KUKA KRL program: EPS_2_251806_MH44A_A_20260212042239.src

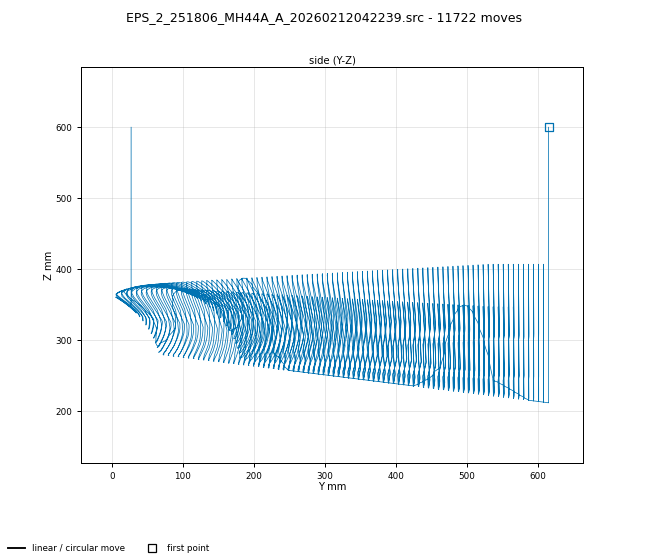
[picture p0: tool path of EPS_2_251806_MH44A_A_20260212042239.src, 11722 of 11724 moves have a stored position in this frame; points joined in program order, loops and branches not executed]
&ACCESS RVP
&REL 4
&COMMENT QRS 19112012
&PARAM EDITMASK = *
DEF PART()
EXT BAS (BAS_COMMAND :IN,REAL :IN )
INT I
BAS (#INITMOV,0 )

;KUKA QRS Post kuka4.cps  Date:22-06-2017 !

File_ID=3016

QRS_PRE_INIT()

;Init var - Until changes are made in qrs_pre_init
Outlet_Square_prg=0
Inlet_1_Square_prg=0
Inlet_2_Square_prg=0
Inlet_3_Square_prg=0
Inlet_4_Square_prg=0
Inlet_5_Square_prg=0

Outlet_1={X 0.000, Y 531.880, Z 306.500, B 0.000, E1 0.000 }
Inlet_1={X 0.000, Y 536.220, Z 246.500, B 0.000, E1 143.000 }
Outlet_1_type=201
Inlet_1_type=201
;QRS#1=Sidecore dimensions
;QRS#2=200-8" PVC SDR 35
;QRS#3=200-8" PVC SDR 35
;QRS#4=
;QRS#5=
;QRS#6=
;QRS#7=
;QRS#8=
;QRS#9=12-08 PSX
;QRS#10=12-08 PSX
;QRS#11=
;QRS#12=
;QRS#13=
;QRS#14=
;QRS#15=
;QRS#16=1220x127x686 2,25'
;QRS#17=EPS Height
;QRS#18=407
;QRS#19=*
;QRS#20= UPDATED VERSION 22-06-2017
;QRS#21=*
Outlet_Square=0100
Inlet_1_Square=0100
Inlet_2_Square=0
Inlet_3_Square=0
Inlet_4_Square=0
Inlet_5_Square=0
Mill_Square=1
Outlet_Square_Prg=204
Inlet_1_Square_prg=204

QRS_INIT()

$ADVANCE=5

; T1
PTP {E1 173.604,E2 173.604}
PTP {X 0,Y 615.501,A -85,B 0,C 180,E1 173.604,E2 173.604,E3 0,E4 0,E5 0,E6 0}
QRS_SPEED_INIT()
LIN {X 0,Y 615.501,Z 600,A -85,B 0,C 180,E1 173.604,E2 173.604,E3 0,E4 0,E5 0,E6 0} C_VEL
LIN {X 0,Y 615.501,Z 221.877,A -85,B 0,C 180,E1 173.604,E2 173.604} C_VEL
LIN {X 0,Y 615.501,Z 213.7,A -85,B 0,C 180,E1 173.604,E2 173.604} C_VEL
LIN {X 0,Y 615.484,Z 211.7,A -85,B 0,C 180,E1 173.418,E2 173.418} C_VEL
LIN {X 0,Y 615.468,Z 211.7,A -85,B 0,C 180,E1 170.802,E2 170.802} C_VEL
LIN {X 0,Y 615.482,Z 211.7,A -85,B 0,C 180,E1 168.14,E2 168.14} C_VEL
LIN {X 0,Y 615.482,Z 211.7,A -85,B 0,C 180,E1 165.452,E2 165.452} C_VEL
LIN {X 0,Y 615.471,Z 211.7,A -85,B 0,C 180,E1 162.73,E2 162.73} C_VEL
LIN {X 0,Y 615.494,Z 212.13,A -85,B 0,C 180,E1 162.045,E2 162.045} C_VEL
LIN {X 0,Y 615.475,Z 215.539,A -85,B 0,C 180,E1 159.27,E2 159.27} C_VEL
LIN {X 0,Y 615.487,Z 218.065,A -85,B 0,C 180,E1 157.157,E2 157.157} C_VEL
LIN {X 0,Y 615.458,Z 220.676,A -85,B 0,C 180,E1 155.008,E2 155.008} C_VEL
LIN {X 0,Y 615.443,Z 223.522,A -85,B 0,C 180,E1 152.822,E2 152.822} C_VEL
LIN {X 0,Y 615.473,Z 226.996,A -85,B 0,C 180,E1 150.206,E2 150.206} C_VEL
LIN {X 0,Y 615.457,Z 230.596,A -85,B 0,C 180,E1 147.542,E2 147.542} C_VEL
LIN {X 0,Y 615.42,Z 233.849,A -85,B 0,C 180,E1 145.182,E2 145.182} C_VEL
LIN {X 0,Y 615.429,Z 237.237,A -85,B 0,C 180,E1 142.756,E2 142.756} C_VEL
LIN {X 0,Y 615.465,Z 241.237,A -85,B 0,C 180,E1 139.912,E2 139.912} C_VEL
LIN {X 0,Y 615.478,Z 243.199,A -85,B 0,C 180,E1 138.54,E2 138.54} C_VEL
LIN {X 0,Y 615.494,Z 257.019,A -85,B 0,C 180,E1 138.227,E2 138.227} C_VEL
LIN {X 0,Y 615.457,Z 268.364,A -85,B 0,C 180,E1 137.852,E2 137.852} C_VEL
LIN {X 0,Y 615.434,Z 280.793,A -85,B 0,C 180,E1 137.3,E2 137.3} C_VEL
LIN {X 0,Y 615.479,Z 291.826,A -85,B 0,C 180,E1 136.662,E2 136.662} C_VEL
LIN {X 0,Y 615.498,Z 302.999,A -85,B 0,C 180,E1 135.854,E2 135.854} C_VEL
LIN {X 0,Y 615.498,Z 311.781,A -85,B 0,C 180,E1 135.067,E2 135.067} C_VEL
LIN {X 0,Y 615.498,Z 320.153,A -85,B 0,C 180,E1 134.148,E2 134.148} C_VEL
LIN {X 0,Y 615.496,Z 328.206,A -85,B 0,C 180,E1 133.051,E2 133.051} C_VEL
LIN {X 0,Y 615.494,Z 333.817,A -85,B 0,C 180,E1 132.083,E2 132.083} C_VEL
LIN {X 0,Y 615.494,Z 338.335,A -85,B 0,C 180,E1 131.098,E2 131.098} C_VEL
LIN {X 0,Y 615.495,Z 341.831,A -85,B 0,C 180,E1 130.092,E2 130.092} C_VEL
LIN {X 0,Y 615.493,Z 344.634,A -85,B 0,C 180,E1 128.903,E2 128.903} C_VEL
LIN {X 0,Y 615.496,Z 345.873,A -85,B 0,C 180,E1 128.016,E2 128.016} C_VEL
LIN {X 0,Y 615.495,Z 346.388,A -85,B 0,C 180,E1 126.94,E2 126.94} C_VEL
LIN {X 0,Y 615.492,Z 345.806,A -85,B 0,C 180,E1 125.837,E2 125.837} C_VEL
LIN {X 0,Y 615.496,Z 344.041,A -85,B 0,C 180,E1 124.705,E2 124.705} C_VEL
LIN {X 0,Y 615.494,Z 340.938,A -85,B 0,C 180,E1 123.538,E2 123.538} C_VEL
LIN {X 0,Y 615.496,Z 336.287,A -85,B 0,C 180,E1 122.335,E2 122.335} C_VEL
LIN {X 0,Y 615.496,Z 331.413,A -85,B 0,C 180,E1 121.387,E2 121.387} C_VEL
LIN {X 0,Y 615.496,Z 324.693,A -85,B 0,C 180,E1 120.348,E2 120.348} C_VEL
LIN {X 0,Y 615.497,Z 317.091,A -85,B 0,C 180,E1 119.405,E2 119.405} C_VEL
LIN {X 0,Y 615.499,Z 307.674,A -85,B 0,C 180,E1 118.456,E2 118.456} C_VEL
LIN {X 0,Y 615.498,Z 297.504,A -85,B 0,C 180,E1 117.636,E2 117.636} C_VEL
LIN {X 0,Y 615.484,Z 286.066,A -85,B 0,C 180,E1 116.897,E2 116.897} C_VEL
LIN {X 0,Y 615.481,Z 274.403,A -85,B 0,C 180,E1 116.307,E2 116.307} C_VEL
LIN {X 0,Y 615.478,Z 262.552,A -85,B 0,C 180,E1 115.852,E2 115.852} C_VEL
LIN {X 0,Y 615.493,Z 249.765,A -85,B 0,C 180,E1 115.501,E2 115.501} C_VEL
LIN {X 0,Y 615.489,Z 243.175,A -85,B 0,C 180,E1 115.355,E2 115.355} C_VEL
LIN {X 0,Y 615.482,Z 239.601,A -85,B 0,C 180,E1 112.844,E2 112.844} C_VEL
LIN {X 0,Y 615.488,Z 235.649,A -85,B 0,C 180,E1 110.032,E2 110.032} C_VEL
LIN {X 0,Y 615.466,Z 231.834,A -85,B 0,C 180,E1 107.27,E2 107.27} C_VEL
LIN {X 0,Y 615.49,Z 228.119,A -85,B 0,C 180,E1 104.548,E2 104.548} C_VEL
LIN {X 0,Y 615.457,Z 224.547,A -85,B 0,C 180,E1 101.861,E2 101.861} C_VEL
LIN {X 0,Y 615.452,Z 221.927,A -85,B 0,C 180,E1 99.862,E2 99.862} C_VEL
LIN {X 0,Y 615.444,Z 219.39,A -85,B 0,C 180,E1 97.875,E2 97.875} C_VEL
LIN {X 0,Y 615.475,Z 216.19,A -85,B 0,C 180,E1 95.241,E2 95.241} C_VEL
LIN {X 0,Y 615.47,Z 212.993,A -85,B 0,C 180,E1 92.617,E2 92.617} C_VEL
LIN {X 0,Y 615.489,Z 211.697,A -85,B 0,C 180,E1 91.308,E2 91.308} C_VEL
LIN {X 0,Y 615.487,Z 211.697,A -85,B 0,C 180,E1 88.691,E2 88.691} C_VEL
LIN {X 0,Y 615.485,Z 211.701,A -85,B 0,C 180,E1 86.071,E2 86.071} C_VEL
LIN {X 0,Y 615.493,Z 211.697,A -85,B 0,C 180,E1 83.402,E2 83.402} C_VEL
LIN {X 0,Y 615.482,Z 211.697,A -85,B 0,C 180,E1 80.8,E2 80.8} C_VEL
LIN {X 0,Y 615.484,Z 211.7,A -85,B 0,C 180,E1 78.138,E2 78.138} C_VEL
LIN {X 0,Y 615.495,Z 211.697,A -85,B 0,C 180,E1 75.45,E2 75.45} C_VEL
LIN {X 0,Y 615.472,Z 211.7,A -85,B 0,C 180,E1 72.728,E2 72.728} C_VEL
LIN {X 0,Y 615.49,Z 211.702,A -85,B 0,C 180,E1 69.967,E2 69.967} C_VEL
LIN {X 0,Y 615.486,Z 211.697,A -85,B 0,C 180,E1 67.155,E2 67.155} C_VEL
LIN {X 0,Y 615.494,Z 211.7,A -85,B 0,C 180,E1 64.284,E2 64.284} C_VEL
LIN {X 0,Y 615.49,Z 211.695,A -85,B 0,C 180,E1 61.341,E2 61.341} C_VEL
LIN {X 0,Y 615.477,Z 211.699,A -85,B 0,C 180,E1 58.912,E2 58.912} C_VEL
LIN {X 0,Y 615.479,Z 211.7,A -85,B 0,C 180,E1 56.464,E2 56.464} C_VEL
LIN {X 0,Y 615.48,Z 211.7,A -85,B 0,C 180,E1 54.165,E2 54.165} C_VEL
LIN {X 0,Y 615.477,Z 211.7,A -85,B 0,C 180,E1 51.93,E2 51.93} C_VEL
LIN {X 0,Y 615.491,Z 211.701,A -85,B 0,C 180,E1 49.393,E2 49.393} C_VEL
LIN {X 0,Y 615.475,Z 211.7,A -85,B 0,C 180,E1 46.753,E2 46.753} C_VEL
LIN {X 0,Y 615.483,Z 211.698,A -85,B 0,C 180,E1 43.996,E2 43.996} C_VEL
LIN {X 0,Y 615.494,Z 211.698,A -85,B 0,C 180,E1 41.471,E2 41.471} C_VEL
LIN {X 0,Y 615.487,Z 211.7,A -85,B 0,C 180,E1 38.902,E2 38.902} C_VEL
LIN {X 0,Y 615.498,Z 211.696,A -85,B 0,C 180,E1 35.834,E2 35.834} C_VEL
LIN {X 0,Y 615.488,Z 211.701,A -85,B 0,C 180,E1 33.234,E2 33.234} C_VEL
LIN {X 0,Y 615.484,Z 211.701,A -85,B 0,C 180,E1 30.918,E2 30.918} C_VEL
LIN {X 0,Y 615.486,Z 211.698,A -85,B 0,C 180,E1 28.449,E2 28.449} C_VEL
LIN {X 0,Y 615.488,Z 211.698,A -85,B 0,C 180,E1 25.568,E2 25.568} C_VEL
LIN {X 0,Y 615.486,Z 211.7,A -85,B 0,C 180,E1 22.843,E2 22.843} C_VEL
LIN {X 0,Y 615.495,Z 211.695,A -85,B 0,C 180,E1 20.031,E2 20.031} C_VEL
LIN {X 0,Y 615.497,Z 211.7,A -85,B 0,C 180,E1 17.269,E2 17.269} C_VEL
LIN {X 0,Y 615.488,Z 211.696,A -85,B 0,C 180,E1 14.548,E2 14.548} C_VEL
LIN {X 0,Y 615.488,Z 211.698,A -85,B 0,C 180,E1 11.86,E2 11.86} C_VEL
LIN {X 0,Y 615.493,Z 211.7,A -85,B 0,C 180,E1 9.198,E2 9.198} C_VEL
LIN {X 0,Y 615.493,Z 211.695,A -85,B 0,C 180,E1 6.555,E2 6.555} C_VEL
LIN {X 0,Y 615.483,Z 211.698,A -85,B 0,C 180,E1 3.927,E2 3.927} C_VEL
LIN {X 0,Y 615.491,Z 211.701,A -85,B 0,C 180,E1 1.308,E2 1.308} C_VEL
LIN {X 0,Y 615.495,Z 211.696,A -85,B 0,C 180,E1 -1.31,E2 -1.31} C_VEL
LIN {X 0,Y 615.477,Z 211.698,A -85,B 0,C 180,E1 -3.93,E2 -3.93} C_VEL
LIN {X 0,Y 615.482,Z 211.701,A -85,B 0,C 180,E1 -6.569,E2 -6.569} C_VEL
LIN {X 0,Y 615.496,Z 211.697,A -85,B 0,C 180,E1 -9.2,E2 -9.2} C_VEL
LIN {X 0,Y 615.47,Z 211.7,A -85,B 0,C 180,E1 -11.862,E2 -11.862} C_VEL
LIN {X 0,Y 615.478,Z 211.701,A -85,B 0,C 180,E1 -14.55,E2 -14.55} C_VEL
LIN {X 0,Y 615.493,Z 211.697,A -85,B 0,C 180,E1 -17.271,E2 -17.271} C_VEL
LIN {X 0,Y 615.47,Z 211.7,A -85,B 0,C 180,E1 -20.034,E2 -20.034} C_VEL
LIN {X 0,Y 615.497,Z 211.699,A -85,B 0,C 180,E1 -22.845,E2 -22.845} C_VEL
LIN {X 0,Y 615.471,Z 211.7,A -85,B 0,C 180,E1 -25.717,E2 -25.717} C_VEL
LIN {X 0,Y 615.494,Z 211.701,A -85,B 0,C 180,E1 -28.45,E2 -28.45} C_VEL
LIN {X 0,Y 615.487,Z 211.697,A -85,B 0,C 180,E1 -31.085,E2 -31.085} C_VEL
LIN {X 0,Y 615.484,Z 211.7,A -85,B 0,C 180,E1 -34.023,E2 -34.023} C_VEL
LIN {X 0,Y 615.49,Z 211.696,A -85,B 0,C 180,E1 -36.936,E2 -36.936} C_VEL
LIN {X 0,Y 615.484,Z 211.7,A -85,B 0,C 180,E1 -39.751,E2 -39.751} C_VEL
LIN {X 0,Y 615.494,Z 211.698,A -85,B 0,C 180,E1 -42.353,E2 -42.353} C_VEL
LIN {X 0,Y 615.483,Z 211.697,A -85,B 0,C 180,E1 -45.07,E2 -45.07} C_VEL
LIN {X 0,Y 615.493,Z 211.701,A -85,B 0,C 180,E1 -47.92,E2 -47.92} C_VEL
LIN {X 0,Y 615.489,Z 211.696,A -85,B 0,C 180,E1 -50.938,E2 -50.938} C_VEL
LIN {X 0,Y 615.486,Z 211.701,A -85,B 0,C 180,E1 -53.574,E2 -53.574} C_VEL
LIN {X 0,Y 615.49,Z 211.764,A -85,B 0,C 180,E1 -54.484,E2 -54.484} C_VEL
LIN {X 0,Y 615.478,Z 220.56,A -85,B 0,C 180,E1 -57.153,E2 -57.153} C_VEL
LIN {X 0,Y 615.476,Z 228.497,A -85,B 0,C 180,E1 -59.46,E2 -59.46} C_VEL
LIN {X 0,Y 615.451,Z 237.756,A -85,B 0,C 180,E1 -62.082,E2 -62.082} C_VEL
LIN {X 0,Y 615.464,Z 247.261,A -85,B 0,C 180,E1 -64.718,E2 -64.718} C_VEL
LIN {X 0,Y 615.448,Z 256.24,A -85,B 0,C 180,E1 -67.153,E2 -67.153} C_VEL
LIN {X 0,Y 615.478,Z 264.815,A -85,B 0,C 180,E1 -69.446,E2 -69.446} C_VEL
LIN {X 0,Y 615.492,Z 276.01,A -85,B 0,C 180,E1 -72.386,E2 -72.386} C_VEL
LIN {X 0,Y 615.484,Z 286.539,A -85,B 0,C 180,E1 -75.112,E2 -75.112} C_VEL
LIN {X 0,Y 615.465,Z 297.082,A -85,B 0,C 180,E1 -77.804,E2 -77.804} C_VEL
LIN {X 0,Y 615.496,Z 299.207,A -85,B 0,C 180,E1 -78.348,E2 -78.348} C_VEL
LIN {X 0,Y 615.497,Z 313.797,A -85,B 0,C 180,E1 -78.64,E2 -78.64} C_VEL
LIN {X 0,Y 615.455,Z 326.947,A -85,B 0,C 180,E1 -79.05,E2 -79.05} C_VEL
LIN {X 0,Y 615.447,Z 338.759,A -85,B 0,C 180,E1 -79.555,E2 -79.555} C_VEL
LIN {X 0,Y 615.497,Z 349.375,A -85,B 0,C 180,E1 -80.137,E2 -80.137} C_VEL
LIN {X 0,Y 615.498,Z 360.223,A -85,B 0,C 180,E1 -80.884,E2 -80.884} C_VEL
LIN {X 0,Y 615.497,Z 370.805,A -85,B 0,C 180,E1 -81.793,E2 -81.793} C_VEL
LIN {X 0,Y 615.498,Z 378.6,A -85,B 0,C 180,E1 -82.619,E2 -82.619} C_VEL
LIN {X 0,Y 615.496,Z 386.198,A -85,B 0,C 180,E1 -83.607,E2 -83.607} C_VEL
LIN {X 0,Y 615.498,Z 393.201,A -85,B 0,C 180,E1 -84.758,E2 -84.758} C_VEL
LIN {X 0,Y 615.494,Z 397.848,A -85,B 0,C 180,E1 -85.743,E2 -85.743} C_VEL
LIN {X 0,Y 615.494,Z 401.397,A -85,B 0,C 180,E1 -86.726,E2 -86.726} C_VEL
LIN {X 0,Y 615.497,Z 403.231,A -85,B 0,C 180,E1 -87.382,E2 -87.382} C_VEL
LIN {X 0,Y 615.5,Z 404.606,A -85,B 0,C 180,E1 -88.036,E2 -88.036} C_VEL
LIN {X 0,Y 615.496,Z 406.173,A -85,B 0,C 180,E1 -89.345,E2 -89.345} C_VEL
LIN {X 0,Y 615.494,Z 406.389,A -85,B 0,C 180,E1 -89.999,E2 -89.999} C_VEL
LIN {X 0,Y 615.495,Z 405.581,A -85,B 0,C 180,E1 -91.308,E2 -91.308} C_VEL
LIN {X 0,Y 615.5,Z 404.609,A -85,B 0,C 180,E1 -91.962,E2 -91.962} C_VEL
LIN {X 0,Y 615.497,Z 403.235,A -85,B 0,C 180,E1 -92.617,E2 -92.617} C_VEL
LIN {X 0,Y 615.496,Z 400.352,A -85,B 0,C 180,E1 -93.6,E2 -93.6} C_VEL
LIN {X 0,Y 615.498,Z 396.444,A -85,B 0,C 180,E1 -94.584,E2 -94.584} C_VEL
LIN {X 0,Y 615.499,Z 391.409,A -85,B 0,C 180,E1 -95.569,E2 -95.569} C_VEL
LIN {X 0,Y 615.497,Z 384.871,A -85,B 0,C 180,E1 -96.583,E2 -96.583} C_VEL
LIN {X 0,Y 615.497,Z 377.139,A -85,B 0,C 180,E1 -97.545,E2 -97.545} C_VEL
LIN {X 0,Y 615.498,Z 369.052,A -85,B 0,C 180,E1 -98.37,E2 -98.37} C_VEL
LIN {X 0,Y 615.499,Z 359.177,A -85,B 0,C 180,E1 -99.198,E2 -99.198} C_VEL
LIN {X 0,Y 615.486,Z 347.993,A -85,B 0,C 180,E1 -99.945,E2 -99.945} C_VEL
LIN {X 0,Y 615.445,Z 337.044,A -85,B 0,C 180,E1 -100.527,E2 -100.527} C_VEL
LIN {X 0,Y 615.461,Z 324.771,A -85,B 0,C 180,E1 -101.031,E2 -101.031} C_VEL
LIN {X 0,Y 615.498,Z 312.093,A -85,B 0,C 180,E1 -101.401,E2 -101.401} C_VEL
LIN {X 0,Y 615.496,Z 299.212,A -85,B 0,C 180,E1 -101.651,E2 -101.651} C_VEL
LIN {X 0,Y 615.469,Z 289.073,A -85,B 0,C 180,E1 -104.24,E2 -104.24} C_VEL
LIN {X 0,Y 615.484,Z 278.644,A -85,B 0,C 180,E1 -106.928,E2 -106.928} C_VEL
LIN {X 0,Y 615.487,Z 268.104,A -85,B 0,C 180,E1 -109.684,E2 -109.684} C_VEL
LIN {X 0,Y 615.474,Z 258.107,A -85,B 0,C 180,E1 -112.342,E2 -112.342} C_VEL
LIN {X 0,Y 615.442,Z 248.325,A -85,B 0,C 180,E1 -114.993,E2 -114.993} C_VEL
LIN {X 0,Y 615.492,Z 239.078,A -85,B 0,C 180,E1 -117.544,E2 -117.544} C_VEL
LIN {X 0,Y 615.459,Z 229.832,A -85,B 0,C 180,E1 -120.161,E2 -120.161} C_VEL
LIN {X 0,Y 615.486,Z 221.872,A -85,B 0,C 180,E1 -122.457,E2 -122.457} C_VEL
LIN {X 0,Y 615.491,Z 212.793,A -85,B 0,C 180,E1 -125.213,E2 -125.213} C_VEL
LIN {X 0,Y 615.486,Z 211.697,A -85,B 0,C 180,E1 -125.615,E2 -125.615} C_VEL
LIN {X 0,Y 615.469,Z 211.7,A -85,B 0,C 180,E1 -128.069,E2 -128.069} C_VEL
LIN {X 0,Y 615.474,Z 211.701,A -85,B 0,C 180,E1 -130.607,E2 -130.607} C_VEL
LIN {X 0,Y 615.499,Z 211.698,A -85,B 0,C 180,E1 -133.243,E2 -133.243} C_VEL
LIN {X 0,Y 615.469,Z 211.7,A -85,B 0,C 180,E1 -136.003,E2 -136.003} C_VEL
LIN {X 0,Y 615.476,Z 211.7,A -85,B 0,C 180,E1 -138.525,E2 -138.525} C_VEL
LIN {X 0,Y 615.494,Z 211.701,A -85,B 0,C 180,E1 -141.095,E2 -141.095} C_VEL
LIN {X 0,Y 615.48,Z 211.7,A -85,B 0,C 180,E1 -143.574,E2 -143.574} C_VEL
LIN {X 0,Y 615.474,Z 211.7,A -85,B 0,C 180,E1 -145.976,E2 -145.976} C_VEL
LIN {X 0,Y 615.472,Z 211.7,A -85,B 0,C 180,E1 -148.313,E2 -148.313} C_VEL
LIN {X 0,Y 615.484,Z 211.697,A -85,B 0,C 180,E1 -150.593,E2 -150.593} C_VEL
LIN {X 0,Y 615.492,Z 211.702,A -85,B 0,C 180,E1 -153.555,E2 -153.555} C_VEL
LIN {X 0,Y 615.485,Z 211.7,A -85,B 0,C 180,E1 -155.99,E2 -155.99} C_VEL
LIN {X 0,Y 615.485,Z 211.697,A -85,B 0,C 180,E1 -158.567,E2 -158.567} C_VEL
LIN {X 0,Y 615.495,Z 211.699,A -85,B 0,C 180,E1 -161.391,E2 -161.391} C_VEL
LIN {X 0,Y 615.478,Z 211.699,A -85,B 0,C 180,E1 -164.094,E2 -164.094} C_VEL
LIN {X 0,Y 615.498,Z 211.695,A -85,B 0,C 180,E1 -166.798,E2 -166.798} C_VEL
LIN {X 0,Y 615.487,Z 211.702,A -85,B 0,C 180,E1 -169.472,E2 -169.472} C_VEL
LIN {X 0,Y 615.479,Z 211.698,A -85,B 0,C 180,E1 -172.123,E2 -172.123} C_VEL
LIN {X 0,Y 615.495,Z 211.696,A -85,B 0,C 180,E1 -174.758,E2 -174.758} C_VEL
LIN {X 0,Y 615.489,Z 211.701,A -85,B 0,C 180,E1 -177.381,E2 -177.381} C_VEL
LIN {X 0,Y 615.482,Z 211.698,A -85,B 0,C 180,E1 -179.999,E2 -179.999} C_VEL
LIN {X 0,Y 615.494,Z 211.695,A -85,B 0,C 180,E1 -182.617,E2 -182.617} C_VEL
LIN {X 0,Y 615.496,Z 211.7,A -85,B 0,C 180,E1 -185.24,E2 -185.24} C_VEL
LIN {X 0,Y 615.484,Z 211.7,A -85,B 0,C 180,E1 -186.582,E2 -186.582} C_VEL
LIN {X 0,Y 614.8,Z 211.847,A -85,B 0,C 180,E1 -187.128,E2 -187.128} C_VEL
LIN {X 0,Y 611.954,Z 212.259,A -85,B 0,C 180,E1 -188.014,E2 -188.014} C_VEL
LIN {X 0,Y 609.562,Z 212.568,A -85,B 0,C 180,E1 -188.727,E2 -188.727} C_VEL
LIN {X 0,Y 608.536,Z 212.685,A -85,B 0,C 180,E1 -189.276,E2 -189.276} C_VEL
LIN {X 0,Y 608.452,Z 212.694,A -85,B 0,C 180,E1 -189.463,E2 -189.463} C_VEL
LIN {X 0,Y 608.458,Z 212.697,A -85,B 0,C 180,E1 -191.999,E2 -191.999} C_VEL
LIN {X 0,Y 608.469,Z 212.693,A -85,B 0,C 180,E1 -194.719,E2 -194.719} C_VEL
LIN {X 0,Y 608.445,Z 212.697,A -85,B 0,C 180,E1 -197.475,E2 -197.475} C_VEL
LIN {X 0,Y 608.42,Z 214.125,A -85,B 0,C 180,E1 -198.869,E2 -198.869} C_VEL
LIN {X 0,Y 608.441,Z 217.534,A -85,B 0,C 180,E1 -201.691,E2 -201.691} C_VEL
LIN {X 0,Y 608.446,Z 220.984,A -85,B 0,C 180,E1 -204.57,E2 -204.57} C_VEL
LIN {X 0,Y 608.391,Z 224.301,A -85,B 0,C 180,E1 -207.193,E2 -207.193} C_VEL
LIN {X 0,Y 608.445,Z 227.967,A -85,B 0,C 180,E1 -209.969,E2 -209.969} C_VEL
LIN {X 0,Y 608.386,Z 231.902,A -85,B 0,C 180,E1 -212.882,E2 -212.882} C_VEL
LIN {X 0,Y 608.375,Z 235.196,A -85,B 0,C 180,E1 -215.28,E2 -215.28} C_VEL
LIN {X 0,Y 608.38,Z 239.308,A -85,B 0,C 180,E1 -218.231,E2 -218.231} C_VEL
LIN {X 0,Y 608.384,Z 242.257,A -85,B 0,C 180,E1 -220.323,E2 -220.323} C_VEL
LIN {X 0,Y 608.398,Z 243.686,A -85,B 0,C 180,E1 -221.33,E2 -221.33} C_VEL
LIN {X 0,Y 608.546,Z 257.819,A -85,B 0,C 180,E1 -221.662,E2 -221.662} C_VEL
LIN {X 0,Y 608.477,Z 269.465,A -85,B 0,C 180,E1 -222.058,E2 -222.058} C_VEL
LIN {X 0,Y 608.448,Z 281.581,A -85,B 0,C 180,E1 -222.614,E2 -222.614} C_VEL
LIN {X 0,Y 608.482,Z 293.339,A -85,B 0,C 180,E1 -223.311,E2 -223.311} C_VEL
LIN {X 0,Y 608.471,Z 303.546,A -85,B 0,C 180,E1 -224.066,E2 -224.066} C_VEL
LIN {X 0,Y 608.458,Z 313.645,A -85,B 0,C 180,E1 -224.999,E2 -224.999} C_VEL
LIN {X 0,Y 608.465,Z 321.852,A -85,B 0,C 180,E1 -225.932,E2 -225.932} C_VEL
LIN {X 0,Y 608.448,Z 328.559,A -85,B 0,C 180,E1 -226.867,E2 -226.867} C_VEL
LIN {X 0,Y 608.429,Z 334.694,A -85,B 0,C 180,E1 -227.937,E2 -227.937} C_VEL
LIN {X 0,Y 608.43,Z 338.727,A -85,B 0,C 180,E1 -228.822,E2 -228.822} C_VEL
LIN {X 0,Y 608.434,Z 343.095,A -85,B 0,C 180,E1 -230.129,E2 -230.129} C_VEL
LIN {X 0,Y 608.414,Z 345.782,A -85,B 0,C 180,E1 -231.409,E2 -231.409} C_VEL
LIN {X 0,Y 608.425,Z 346.691,A -85,B 0,C 180,E1 -232.251,E2 -232.251} C_VEL
LIN {X 0,Y 608.43,Z 346.997,A -85,B 0,C 180,E1 -233.084,E2 -233.084} C_VEL
LIN {X 0,Y 608.441,Z 346.611,A -85,B 0,C 180,E1 -233.953,E2 -233.953} C_VEL
LIN {X 0,Y 608.423,Z 345.094,A -85,B 0,C 180,E1 -235.095,E2 -235.095} C_VEL
LIN {X 0,Y 608.434,Z 342.044,A -85,B 0,C 180,E1 -236.328,E2 -236.328} C_VEL
LIN {X 0,Y 608.428,Z 337.821,A -85,B 0,C 180,E1 -237.479,E2 -237.479} C_VEL
LIN {X 0,Y 608.444,Z 331.846,A -85,B 0,C 180,E1 -238.683,E2 -238.683} C_VEL
LIN {X 0,Y 608.444,Z 324.771,A -85,B 0,C 180,E1 -239.772,E2 -239.772} C_VEL
LIN {X 0,Y 608.45,Z 316.476,A -85,B 0,C 180,E1 -240.791,E2 -240.791} C_VEL
LIN {X 0,Y 608.467,Z 306.911,A -85,B 0,C 180,E1 -241.735,E2 -241.735} C_VEL
LIN {X 0,Y 608.493,Z 296.237,A -85,B 0,C 180,E1 -242.58,E2 -242.58} C_VEL
LIN {X 0,Y 608.481,Z 286.114,A -85,B 0,C 180,E1 -243.228,E2 -243.228} C_VEL
LIN {X 0,Y 608.494,Z 274.258,A -85,B 0,C 180,E1 -243.829,E2 -243.829} C_VEL
LIN {X 0,Y 608.522,Z 261.978,A -85,B 0,C 180,E1 -244.3,E2 -244.3} C_VEL
LIN {X 0,Y 608.536,Z 249.165,A -85,B 0,C 180,E1 -244.648,E2 -244.648} C_VEL
LIN {X 0,Y 608.422,Z 243.676,A -85,B 0,C 180,E1 -244.767,E2 -244.767} C_VEL
LIN {X 0,Y 608.416,Z 239.68,A -85,B 0,C 180,E1 -247.593,E2 -247.593} C_VEL
LIN {X 0,Y 608.402,Z 235.722,A -85,B 0,C 180,E1 -250.428,E2 -250.428} C_VEL
LIN {X 0,Y 608.436,Z 231.888,A -85,B 0,C 180,E1 -253.216,E2 -253.216} C_VEL
LIN {X 0,Y 608.421,Z 228.138,A -85,B 0,C 180,E1 -255.994,E2 -255.994} C_VEL
LIN {X 0,Y 608.395,Z 224.591,A -85,B 0,C 180,E1 -258.675,E2 -258.675} C_VEL
LIN {X 0,Y 608.454,Z 221.141,A -85,B 0,C 180,E1 -261.365,E2 -261.365} C_VEL
LIN {X 0,Y 608.381,Z 217.909,A -85,B 0,C 180,E1 -264.033,E2 -264.033} C_VEL
LIN {X 0,Y 608.435,Z 214.682,A -85,B 0,C 180,E1 -266.69,E2 -266.69} C_VEL
LIN {X 0,Y 608.439,Z 213.067,A -85,B 0,C 180,E1 -268.015,E2 -268.015} C_VEL
LIN {X 0,Y 608.484,Z 212.693,A -85,B 0,C 180,E1 -269.339,E2 -269.339} C_VEL
LIN {X 0,Y 608.451,Z 212.696,A -85,B 0,C 180,E1 -271.986,E2 -271.986} C_VEL
LIN {X 0,Y 608.448,Z 212.695,A -85,B 0,C 180,E1 -274.638,E2 -274.638} C_VEL
LIN {X 0,Y 608.48,Z 212.693,A -85,B 0,C 180,E1 -277.3,E2 -277.3} C_VEL
LIN {X 0,Y 608.458,Z 212.695,A -85,B 0,C 180,E1 -279.978,E2 -279.978} C_VEL
LIN {X 0,Y 608.477,Z 212.692,A -85,B 0,C 180,E1 -282.678,E2 -282.678} C_VEL
LIN {X 0,Y 608.468,Z 212.696,A -85,B 0,C 180,E1 -285.407,E2 -285.407} C_VEL
LIN {X 0,Y 608.451,Z 212.695,A -85,B 0,C 180,E1 -288.172,E2 -288.172} C_VEL
LIN {X 0,Y 608.455,Z 212.696,A -85,B 0,C 180,E1 -290.982,E2 -290.982} C_VEL
LIN {X 0,Y 608.448,Z 212.696,A -85,B 0,C 180,E1 -293.125,E2 -293.125} C_VEL
LIN {X 0,Y 608.451,Z 212.696,A -85,B 0,C 180,E1 -296.036,E2 -296.036} C_VEL
LIN {X 0,Y 608.477,Z 212.692,A -85,B 0,C 180,E1 -298.624,E2 -298.624} C_VEL
LIN {X 0,Y 608.468,Z 212.694,A -85,B 0,C 180,E1 -301.317,E2 -301.317} C_VEL
LIN {X 0,Y 608.468,Z 212.696,A -85,B 0,C 180,E1 -303.737,E2 -303.737} C_VEL
LIN {X 0,Y 608.471,Z 212.696,A -85,B 0,C 180,E1 -306.091,E2 -306.091} C_VEL
LIN {X 0,Y 608.456,Z 212.696,A -85,B 0,C 180,E1 -308.59,E2 -308.59} C_VEL
LIN {X 0,Y 608.45,Z 212.695,A -85,B 0,C 180,E1 -311.343,E2 -311.343} C_VEL
LIN {X 0,Y 608.465,Z 212.695,A -85,B 0,C 180,E1 -314.267,E2 -314.267} C_VEL
LIN {X 0,Y 608.436,Z 212.697,A -85,B 0,C 180,E1 -317.041,E2 -317.041} C_VEL
LIN {X 0,Y 608.45,Z 212.697,A -85,B 0,C 180,E1 -319.698,E2 -319.698} C_VEL
LIN {X 0,Y 608.462,Z 212.696,A -85,B 0,C 180,E1 -322.255,E2 -322.255} C_VEL
LIN {X 0,Y 608.442,Z 212.697,A -85,B 0,C 180,E1 -324.724,E2 -324.724} C_VEL
LIN {X 0,Y 608.455,Z 212.695,A -85,B 0,C 180,E1 -327.122,E2 -327.122} C_VEL
LIN {X 0,Y 608.47,Z 212.695,A -85,B 0,C 180,E1 -330.029,E2 -330.029} C_VEL
LIN {X 0,Y 608.467,Z 212.693,A -85,B 0,C 180,E1 -332.796,E2 -332.796} C_VEL
LIN {X 0,Y 608.449,Z 212.695,A -85,B 0,C 180,E1 -335.43,E2 -335.43} C_VEL
LIN {X 0,Y 608.464,Z 212.695,A -85,B 0,C 180,E1 -338.31,E2 -338.31} C_VEL
LIN {X 0,Y 608.454,Z 212.695,A -85,B 0,C 180,E1 -341.132,E2 -341.132} C_VEL
LIN {X 0,Y 608.456,Z 212.697,A -85,B 0,C 180,E1 -343.907,E2 -343.907} C_VEL
LIN {X 0,Y 608.455,Z 212.694,A -85,B 0,C 180,E1 -346.645,E2 -346.645} C_VEL
LIN {X 0,Y 608.463,Z 212.695,A -85,B 0,C 180,E1 -349.351,E2 -349.351} C_VEL
LIN {X 0,Y 608.473,Z 212.694,A -85,B 0,C 180,E1 -352.034,E2 -352.034} C_VEL
LIN {X 0,Y 608.451,Z 212.695,A -85,B 0,C 180,E1 -354.699,E2 -354.699} C_VEL
LIN {X 0,Y 608.478,Z 212.693,A -85,B 0,C 180,E1 -357.353,E2 -357.353} C_VEL
LIN {X 0,Y 608.478,Z 212.694,A -85,B 0,C 180,E1 -360.001,E2 -360.001} C_VEL
LIN {X 0,Y 608.465,Z 212.693,A -85,B 0,C 180,E1 -362.649,E2 -362.649} C_VEL
LIN {X 0,Y 608.466,Z 212.694,A -85,B 0,C 180,E1 -365.303,E2 -365.303} C_VEL
LIN {X 0,Y 608.479,Z 212.694,A -85,B 0,C 180,E1 -367.968,E2 -367.968} C_VEL
LIN {X 0,Y 608.451,Z 212.695,A -85,B 0,C 180,E1 -370.651,E2 -370.651} C_VEL
LIN {X 0,Y 608.469,Z 212.694,A -85,B 0,C 180,E1 -373.357,E2 -373.357} C_VEL
LIN {X 0,Y 608.456,Z 212.696,A -85,B 0,C 180,E1 -376.095,E2 -376.095} C_VEL
LIN {X 0,Y 608.456,Z 212.694,A -85,B 0,C 180,E1 -378.87,E2 -378.87} C_VEL
LIN {X 0,Y 608.469,Z 212.695,A -85,B 0,C 180,E1 -381.692,E2 -381.692} C_VEL
LIN {X 0,Y 608.451,Z 212.695,A -85,B 0,C 180,E1 -384.572,E2 -384.572} C_VEL
LIN {X 0,Y 608.489,Z 212.692,A -85,B 0,C 180,E1 -387.208,E2 -387.208} C_VEL
LIN {X 0,Y 608.445,Z 212.696,A -85,B 0,C 180,E1 -389.967,E2 -389.967} C_VEL
LIN {X 0,Y 608.453,Z 212.695,A -85,B 0,C 180,E1 -392.52,E2 -392.52} C_VEL
LIN {X 0,Y 608.442,Z 212.699,A -85,B 0,C 180,E1 -395.278,E2 -395.278} C_VEL
LIN {X 0,Y 608.463,Z 212.696,A -85,B 0,C 180,E1 -397.747,E2 -397.747} C_VEL
LIN {X 0,Y 608.451,Z 212.695,A -85,B 0,C 180,E1 -400.328,E2 -400.328} C_VEL
LIN {X 0,Y 608.482,Z 212.694,A -85,B 0,C 180,E1 -403.309,E2 -403.309} C_VEL
LIN {X 0,Y 608.465,Z 212.693,A -85,B 0,C 180,E1 -406.129,E2 -406.129} C_VEL
LIN {X 0,Y 608.464,Z 212.694,A -85,B 0,C 180,E1 -408.823,E2 -408.823} C_VEL
LIN {X 0,Y 608.457,Z 212.695,A -85,B 0,C 180,E1 -411.762,E2 -411.762} C_VEL
LIN {X 0,Y 608.476,Z 212.766,A -85,B 0,C 180,E1 -414.317,E2 -414.317} C_VEL
LIN {X 0,Y 608.521,Z 220.56,A -85,B 0,C 180,E1 -416.729,E2 -416.729} C_VEL
LIN {X 0,Y 608.502,Z 229.822,A -85,B 0,C 180,E1 -419.456,E2 -419.456} C_VEL
LIN {X 0,Y 608.469,Z 239.125,A -85,B 0,C 180,E1 -422.109,E2 -422.109} C_VEL
LIN {X 0,Y 608.454,Z 248.392,A -85,B 0,C 180,E1 -424.698,E2 -424.698} C_VEL
LIN {X 0,Y 608.465,Z 258.723,A -85,B 0,C 180,E1 -427.523,E2 -427.523} C_VEL
LIN {X 0,Y 608.457,Z 269.574,A -85,B 0,C 180,E1 -430.429,E2 -430.429} C_VEL
LIN {X 0,Y 608.452,Z 280.166,A -85,B 0,C 180,E1 -433.215,E2 -433.215} C_VEL
LIN {X 0,Y 608.443,Z 290.884,A -85,B 0,C 180,E1 -435.994,E2 -435.994} C_VEL
LIN {X 0,Y 608.443,Z 299.528,A -85,B 0,C 180,E1 -438.211,E2 -438.211} C_VEL
LIN {X 0,Y 608.545,Z 314.673,A -85,B 0,C 180,E1 -438.529,E2 -438.529} C_VEL
LIN {X 0,Y 608.478,Z 327.497,A -85,B 0,C 180,E1 -438.939,E2 -438.939} C_VEL
LIN {X 0,Y 608.474,Z 338.908,A -85,B 0,C 180,E1 -439.434,E2 -439.434} C_VEL
LIN {X 0,Y 608.486,Z 349.568,A -85,B 0,C 180,E1 -440.023,E2 -440.023} C_VEL
LIN {X 0,Y 608.483,Z 360.466,A -85,B 0,C 180,E1 -440.778,E2 -440.778} C_VEL
LIN {X 0,Y 608.475,Z 371.105,A -85,B 0,C 180,E1 -441.698,E2 -441.698} C_VEL
LIN {X 0,Y 608.471,Z 378.955,A -85,B 0,C 180,E1 -442.533,E2 -442.533} C_VEL
LIN {X 0,Y 608.461,Z 386.285,A -85,B 0,C 180,E1 -443.484,E2 -443.484} C_VEL
LIN {X 0,Y 608.451,Z 391.862,A -85,B 0,C 180,E1 -444.365,E2 -444.365} C_VEL
LIN {X 0,Y 608.432,Z 396.947,A -85,B 0,C 180,E1 -445.362,E2 -445.362} C_VEL
LIN {X 0,Y 608.449,Z 400.894,A -85,B 0,C 180,E1 -446.357,E2 -446.357} C_VEL
LIN {X 0,Y 608.425,Z 403.807,A -85,B 0,C 180,E1 -447.351,E2 -447.351} C_VEL
LIN {X 0,Y 608.445,Z 405.2,A -85,B 0,C 180,E1 -448.014,E2 -448.014} C_VEL
LIN {X 0,Y 608.438,Z 406.783,A -85,B 0,C 180,E1 -449.338,E2 -449.338} C_VEL
LIN {X 0,Y 608.434,Z 407,A -85,B 0,C 180,E1 -449.999,E2 -449.999} C_VEL
LIN {X 0,Y 608.448,Z 406.185,A -85,B 0,C 180,E1 -451.323,E2 -451.323} C_VEL
LIN {X 0,Y 608.445,Z 405.202,A -85,B 0,C 180,E1 -451.985,E2 -451.985} C_VEL
LIN {X 0,Y 608.425,Z 403.811,A -85,B 0,C 180,E1 -452.648,E2 -452.648} C_VEL
LIN {X 0,Y 608.449,Z 400.898,A -85,B 0,C 180,E1 -453.642,E2 -453.642} C_VEL
LIN {X 0,Y 608.432,Z 396.953,A -85,B 0,C 180,E1 -454.637,E2 -454.637} C_VEL
LIN {X 0,Y 608.438,Z 390.881,A -85,B 0,C 180,E1 -455.8,E2 -455.8} C_VEL
LIN {X 0,Y 608.462,Z 384.24,A -85,B 0,C 180,E1 -456.799,E2 -456.799} C_VEL
LIN {X 0,Y 608.456,Z 375.995,A -85,B 0,C 180,E1 -457.8,E2 -457.8} C_VEL
LIN {X 0,Y 608.472,Z 367.544,A -85,B 0,C 180,E1 -458.635,E2 -458.635} C_VEL
LIN {X 0,Y 608.481,Z 357.1,A -85,B 0,C 180,E1 -459.473,E2 -459.473} C_VEL
LIN {X 0,Y 608.494,Z 346.767,A -85,B 0,C 180,E1 -460.144,E2 -460.144} C_VEL
LIN {X 0,Y 608.469,Z 335.851,A -85,B 0,C 180,E1 -460.713,E2 -460.713} C_VEL
LIN {X 0,Y 608.493,Z 324.095,A -85,B 0,C 180,E1 -461.186,E2 -461.186} C_VEL
LIN {X 0,Y 608.549,Z 311.297,A -85,B 0,C 180,E1 -461.554,E2 -461.554} C_VEL
LIN {X 0,Y 608.443,Z 299.533,A -85,B 0,C 180,E1 -461.788,E2 -461.788} C_VEL
LIN {X 0,Y 608.435,Z 289.438,A -85,B 0,C 180,E1 -464.379,E2 -464.379} C_VEL
LIN {X 0,Y 608.442,Z 278.847,A -85,B 0,C 180,E1 -467.13,E2 -467.13} C_VEL
LIN {X 0,Y 608.457,Z 269.58,A -85,B 0,C 180,E1 -469.57,E2 -469.57} C_VEL
LIN {X 0,Y 608.46,Z 258.728,A -85,B 0,C 180,E1 -472.476,E2 -472.476} C_VEL
LIN {X 0,Y 608.454,Z 248.398,A -85,B 0,C 180,E1 -475.3,E2 -475.3} C_VEL
LIN {X 0,Y 608.468,Z 239.13,A -85,B 0,C 180,E1 -477.89,E2 -477.89} C_VEL
LIN {X 0,Y 608.482,Z 229.784,A -85,B 0,C 180,E1 -480.543,E2 -480.543} C_VEL
LIN {X 0,Y 608.519,Z 221.841,A -85,B 0,C 180,E1 -482.875,E2 -482.875} C_VEL
LIN {X 0,Y 608.551,Z 214.1,A -85,B 0,C 180,E1 -485.27,E2 -485.27} C_VEL
LIN {X 0,Y 608.472,Z 212.694,A -85,B 0,C 180,E1 -485.771,E2 -485.771} C_VEL
LIN {X 0,Y 608.466,Z 212.697,A -85,B 0,C 180,E1 -488.587,E2 -488.587} C_VEL
LIN {X 0,Y 608.469,Z 212.693,A -85,B 0,C 180,E1 -491.342,E2 -491.342} C_VEL
LIN {X 0,Y 608.457,Z 212.698,A -85,B 0,C 180,E1 -494.263,E2 -494.263} C_VEL
LIN {X 0,Y 608.458,Z 212.694,A -85,B 0,C 180,E1 -497.04,E2 -497.04} C_VEL
LIN {X 0,Y 608.458,Z 212.695,A -85,B 0,C 180,E1 -499.696,E2 -499.696} C_VEL
LIN {X 0,Y 608.466,Z 212.696,A -85,B 0,C 180,E1 -502.253,E2 -502.253} C_VEL
LIN {X 0,Y 608.485,Z 212.691,A -85,B 0,C 180,E1 -505.088,E2 -505.088} C_VEL
LIN {X 0,Y 608.463,Z 212.697,A -85,B 0,C 180,E1 -507.905,E2 -507.905} C_VEL
LIN {X 0,Y 608.471,Z 212.693,A -85,B 0,C 180,E1 -510.98,E2 -510.98} C_VEL
LIN {X 0,Y 608.458,Z 212.695,A -85,B 0,C 180,E1 -513.225,E2 -513.225} C_VEL
LIN {X 0,Y 608.461,Z 212.694,A -85,B 0,C 180,E1 -516.154,E2 -516.154} C_VEL
LIN {X 0,Y 608.459,Z 212.696,A -85,B 0,C 180,E1 -519.018,E2 -519.018} C_VEL
LIN {X 0,Y 608.439,Z 212.697,A -85,B 0,C 180,E1 -521.827,E2 -521.827} C_VEL
LIN {X 0,Y 608.474,Z 212.693,A -85,B 0,C 180,E1 -524.593,E2 -524.593} C_VEL
LIN {X 0,Y 608.47,Z 212.694,A -85,B 0,C 180,E1 -527.322,E2 -527.322} C_VEL
LIN {X 0,Y 608.446,Z 212.696,A -85,B 0,C 180,E1 -530.022,E2 -530.022} C_VEL
LIN {X 0,Y 608.484,Z 212.693,A -85,B 0,C 180,E1 -532.7,E2 -532.7} C_VEL
LIN {X 0,Y 608.444,Z 212.697,A -85,B 0,C 180,E1 -535.361,E2 -535.361} C_VEL
LIN {X 0,Y 608.48,Z 212.695,A -85,B 0,C 180,E1 -537.351,E2 -537.351} C_VEL
LIN {X 0,Y 608.472,Z 212.693,A -85,B 0,C 180,E1 -539.999,E2 -539.999} C_VEL
LIN {X 0,Y 608.483,Z 212.691,A -85,B 0,C 180,E1 -542.647,E2 -542.647} C_VEL
LIN {X 0,Y 608.472,Z 212.696,A -85,B 0,C 180,E1 -545.301,E2 -545.301} C_VEL
LIN {X 0,Y 608.477,Z 212.692,A -85,B 0,C 180,E1 -547.966,E2 -547.966} C_VEL
LIN {X 0,Y 608.452,Z 212.694,A -85,B 0,C 180,E1 -549.463,E2 -549.463} C_VEL
LIN {X 0,Y 607.784,Z 212.78,A -85,B 0,C 180,E1 -550.015,E2 -550.015} C_VEL
LIN {X 0,Y 604.93,Z 213.137,A -85,B 0,C 180,E1 -550.912,E2 -550.912} C_VEL
LIN {X 0,Y 602.522,Z 213.437,A -85,B 0,C 180,E1 -551.634,E2 -551.634} C_VEL
LIN {X 0,Y 601.49,Z 213.564,A -85,B 0,C 180,E1 -552.19,E2 -552.19} C_VEL
LIN {X 0,Y 601.407,Z 213.573,A -85,B 0,C 180,E1 -552.379,E2 -552.379} C_VEL
LIN {X 0,Y 601.424,Z 213.57,A -85,B 0,C 180,E1 -554.896,E2 -554.896} C_VEL
LIN {X 0,Y 601.427,Z 213.571,A -85,B 0,C 180,E1 -556.985,E2 -556.985} C_VEL
LIN {X 0,Y 601.39,Z 213.578,A -85,B 0,C 180,E1 -557.687,E2 -557.687} C_VEL
LIN {X 0,Y 601.364,Z 215.039,A -85,B 0,C 180,E1 -559.099,E2 -559.099} C_VEL
LIN {X 0,Y 601.359,Z 218.47,A -85,B 0,C 180,E1 -561.96,E2 -561.96} C_VEL
LIN {X 0,Y 601.384,Z 221.245,A -85,B 0,C 180,E1 -564.283,E2 -564.283} C_VEL
LIN {X 0,Y 601.304,Z 224.625,A -85,B 0,C 180,E1 -567.117,E2 -567.117} C_VEL
LIN {X 0,Y 601.31,Z 227.596,A -85,B 0,C 180,E1 -569.397,E2 -569.397} C_VEL
LIN {X 0,Y 601.302,Z 230.691,A -85,B 0,C 180,E1 -571.731,E2 -571.731} C_VEL
LIN {X 0,Y 601.293,Z 233.918,A -85,B 0,C 180,E1 -574.125,E2 -574.125} C_VEL
LIN {X 0,Y 601.277,Z 237.288,A -85,B 0,C 180,E1 -576.59,E2 -576.59} C_VEL
LIN {X 0,Y 601.295,Z 241.349,A -85,B 0,C 180,E1 -579.52,E2 -579.52} C_VEL
LIN {X 0,Y 601.303,Z 243.68,A -85,B 0,C 180,E1 -581.185,E2 -581.185} C_VEL
LIN {X 0,Y 601.594,Z 248.979,A -85,B 0,C 180,E1 -581.302,E2 -581.302} C_VEL
LIN {X 0,Y 601.551,Z 261.647,A -85,B 0,C 180,E1 -581.647,E2 -581.647} C_VEL
LIN {X 0,Y 601.47,Z 273.415,A -85,B 0,C 180,E1 -582.097,E2 -582.097} C_VEL
LIN {X 0,Y 601.449,Z 284.785,A -85,B 0,C 180,E1 -582.665,E2 -582.665} C_VEL
LIN {X 0,Y 601.477,Z 295.519,A -85,B 0,C 180,E1 -583.346,E2 -583.346} C_VEL
LIN {X 0,Y 601.434,Z 305.897,A -85,B 0,C 180,E1 -584.164,E2 -584.164} C_VEL
LIN {X 0,Y 601.418,Z 315.784,A -85,B 0,C 180,E1 -585.13,E2 -585.13} C_VEL
LIN {X 0,Y 601.376,Z 324.333,A -85,B 0,C 180,E1 -586.179,E2 -586.179} C_VEL
LIN {X 0,Y 601.368,Z 331.771,A -85,B 0,C 180,E1 -587.327,E2 -587.327} C_VEL
LIN {X 0,Y 601.359,Z 337.2,A -85,B 0,C 180,E1 -588.411,E2 -588.411} C_VEL
LIN {X 0,Y 601.325,Z 341.135,A -85,B 0,C 180,E1 -589.434,E2 -589.434} C_VEL
LIN {X 0,Y 601.318,Z 344.06,A -85,B 0,C 180,E1 -590.476,E2 -590.476} C_VEL
LIN {X 0,Y 601.328,Z 346.208,A -85,B 0,C 180,E1 -591.726,E2 -591.726} C_VEL
LIN {X 0,Y 601.351,Z 346.909,A -85,B 0,C 180,E1 -592.626,E2 -592.626} C_VEL
LIN {X 0,Y 601.327,Z 346.762,A -85,B 0,C 180,E1 -593.746,E2 -593.746} C_VEL
LIN {X 0,Y 601.334,Z 345.186,A -85,B 0,C 180,E1 -595.064,E2 -595.064} C_VEL
LIN {X 0,Y 601.323,Z 342.881,A -85,B 0,C 180,E1 -596.077,E2 -596.077} C_VEL
LIN {X 0,Y 601.355,Z 338.834,A -85,B 0,C 180,E1 -597.291,E2 -597.291} C_VEL
LIN {X 0,Y 601.364,Z 334.41,A -85,B 0,C 180,E1 -598.272,E2 -598.272} C_VEL
LIN {X 0,Y 601.38,Z 328.844,A -85,B 0,C 180,E1 -599.252,E2 -599.252} C_VEL
LIN {X 0,Y 601.393,Z 322.017,A -85,B 0,C 180,E1 -600.221,E2 -600.221} C_VEL
LIN {X 0,Y 601.393,Z 313.368,A -85,B 0,C 180,E1 -601.215,E2 -601.215} C_VEL
LIN {X 0,Y 601.446,Z 303.484,A -85,B 0,C 180,E1 -602.135,E2 -602.135} C_VEL
LIN {X 0,Y 601.475,Z 293.379,A -85,B 0,C 180,E1 -602.891,E2 -602.891} C_VEL
LIN {X 0,Y 601.5,Z 282.502,A -85,B 0,C 180,E1 -603.548,E2 -603.548} C_VEL
LIN {X 0,Y 601.518,Z 270.739,A -85,B 0,C 180,E1 -604.108,E2 -604.108} C_VEL
LIN {X 0,Y 601.577,Z 258.172,A -85,B 0,C 180,E1 -604.552,E2 -604.552} C_VEL
LIN {X 0,Y 601.473,Z 244.911,A -85,B 0,C 180,E1 -604.871,E2 -604.871} C_VEL
LIN {X 0,Y 601.323,Z 243.671,A -85,B 0,C 180,E1 -604.911,E2 -604.911} C_VEL
LIN {X 0,Y 601.361,Z 240.187,A -85,B 0,C 180,E1 -607.403,E2 -607.403} C_VEL
LIN {X 0,Y 601.307,Z 236.342,A -85,B 0,C 180,E1 -610.188,E2 -610.188} C_VEL
LIN {X 0,Y 601.34,Z 232.498,A -85,B 0,C 180,E1 -613.012,E2 -613.012} C_VEL
LIN {X 0,Y 601.328,Z 228.592,A -85,B 0,C 180,E1 -615.937,E2 -615.937} C_VEL
LIN {X 0,Y 601.302,Z 225.186,A -85,B 0,C 180,E1 -618.54,E2 -618.54} C_VEL
LIN {X 0,Y 601.373,Z 221.843,A -85,B 0,C 180,E1 -621.262,E2 -621.262} C_VEL
LIN {X 0,Y 601.326,Z 218.577,A -85,B 0,C 180,E1 -623.963,E2 -623.963} C_VEL
LIN {X 0,Y 601.355,Z 215.32,A -85,B 0,C 180,E1 -626.651,E2 -626.651} C_VEL
LIN {X 0,Y 601.385,Z 213.708,A -85,B 0,C 180,E1 -627.992,E2 -627.992} C_VEL
LIN {X 0,Y 601.429,Z 213.57,A -85,B 0,C 180,E1 -630.001,E2 -630.001} C_VEL
LIN {X 0,Y 601.433,Z 213.57,A -85,B 0,C 180,E1 -632.68,E2 -632.68} C_VEL
LIN {X 0,Y 601.428,Z 213.571,A -85,B 0,C 180,E1 -635.365,E2 -635.365} C_VEL
LIN {X 0,Y 601.429,Z 213.569,A -85,B 0,C 180,E1 -638.062,E2 -638.062} C_VEL
LIN {X 0,Y 601.42,Z 213.573,A -85,B 0,C 180,E1 -641.019,E2 -641.019} C_VEL
LIN {X 0,Y 601.416,Z 213.572,A -85,B 0,C 180,E1 -643.517,E2 -643.517} C_VEL
LIN {X 0,Y 601.429,Z 213.57,A -85,B 0,C 180,E1 -646.288,E2 -646.288} C_VEL
LIN {X 0,Y 601.409,Z 213.574,A -85,B 0,C 180,E1 -649.1,E2 -649.1} C_VEL
LIN {X 0,Y 601.402,Z 213.576,A -85,B 0,C 180,E1 -651.24,E2 -651.24} C_VEL
LIN {X 0,Y 601.414,Z 213.574,A -85,B 0,C 180,E1 -653.411,E2 -653.411} C_VEL
LIN {X 0,Y 601.405,Z 213.572,A -85,B 0,C 180,E1 -656.364,E2 -656.364} C_VEL
LIN {X 0,Y 601.439,Z 213.569,A -85,B 0,C 180,E1 -658.793,E2 -658.793} C_VEL
LIN {X 0,Y 601.41,Z 213.573,A -85,B 0,C 180,E1 -661.727,E2 -661.727} C_VEL
LIN {X 0,Y 601.428,Z 213.57,A -85,B 0,C 180,E1 -664.119,E2 -664.119} C_VEL
LIN {X 0,Y 601.41,Z 213.572,A -85,B 0,C 180,E1 -666.583,E2 -666.583} C_VEL
LIN {X 0,Y 601.433,Z 213.572,A -85,B 0,C 180,E1 -669.537,E2 -669.537} C_VEL
LIN {X 0,Y 601.434,Z 213.57,A -85,B 0,C 180,E1 -672.669,E2 -672.669} C_VEL
LIN {X 0,Y 601.42,Z 213.572,A -85,B 0,C 180,E1 -675.484,E2 -675.484} C_VEL
LIN {X 0,Y 601.425,Z 213.571,A -85,B 0,C 180,E1 -678.408,E2 -678.408} C_VEL
LIN {X 0,Y 601.437,Z 213.571,A -85,B 0,C 180,E1 -680.877,E2 -680.877} C_VEL
LIN {X 0,Y 601.442,Z 213.568,A -85,B 0,C 180,E1 -683.735,E2 -683.735} C_VEL
LIN {X 0,Y 601.429,Z 213.573,A -85,B 0,C 180,E1 -686.688,E2 -686.688} C_VEL
LIN {X 0,Y 601.414,Z 213.574,A -85,B 0,C 180,E1 -689.059,E2 -689.059} C_VEL
LIN {X 0,Y 601.435,Z 213.571,A -85,B 0,C 180,E1 -691.375,E2 -691.375} C_VEL
LIN {X 0,Y 601.414,Z 213.571,A -85,B 0,C 180,E1 -694.134,E2 -694.134} C_VEL
LIN {X 0,Y 601.396,Z 213.574,A -85,B 0,C 180,E1 -696.59,E2 -696.59} C_VEL
LIN {X 0,Y 601.436,Z 213.57,A -85,B 0,C 180,E1 -699.48,E2 -699.48} C_VEL
LIN {X 0,Y 601.4,Z 213.574,A -85,B 0,C 180,E1 -702.313,E2 -702.313} C_VEL
LIN {X 0,Y 601.41,Z 213.572,A -85,B 0,C 180,E1 -704.41,E2 -704.41} C_VEL
LIN {X 0,Y 601.422,Z 213.573,A -85,B 0,C 180,E1 -707.173,E2 -707.173} C_VEL
LIN {X 0,Y 601.428,Z 213.57,A -85,B 0,C 180,E1 -709.906,E2 -709.906} C_VEL
LIN {X 0,Y 601.412,Z 213.572,A -85,B 0,C 180,E1 -712.616,E2 -712.616} C_VEL
LIN {X 0,Y 601.429,Z 213.573,A -85,B 0,C 180,E1 -715.309,E2 -715.309} C_VEL
LIN {X 0,Y 601.414,Z 213.572,A -85,B 0,C 180,E1 -717.992,E2 -717.992} C_VEL
LIN {X 0,Y 601.441,Z 213.569,A -85,B 0,C 180,E1 -720.671,E2 -720.671} C_VEL
LIN {X 0,Y 601.433,Z 213.572,A -85,B 0,C 180,E1 -723.351,E2 -723.351} C_VEL
LIN {X 0,Y 601.404,Z 213.573,A -85,B 0,C 180,E1 -726.038,E2 -726.038} C_VEL
LIN {X 0,Y 601.442,Z 213.57,A -85,B 0,C 180,E1 -728.062,E2 -728.062} C_VEL
LIN {X 0,Y 601.422,Z 213.571,A -85,B 0,C 180,E1 -731.007,E2 -731.007} C_VEL
LIN {X 0,Y 601.415,Z 213.574,A -85,B 0,C 180,E1 -733.517,E2 -733.517} C_VEL
LIN {X 0,Y 601.434,Z 213.569,A -85,B 0,C 180,E1 -736.288,E2 -736.288} C_VEL
LIN {X 0,Y 601.421,Z 213.572,A -85,B 0,C 180,E1 -739.1,E2 -739.1} C_VEL
LIN {X 0,Y 601.413,Z 213.572,A -85,B 0,C 180,E1 -741.24,E2 -741.24} C_VEL
LIN {X 0,Y 601.432,Z 213.57,A -85,B 0,C 180,E1 -744.142,E2 -744.142} C_VEL
LIN {X 0,Y 601.461,Z 213.567,A -85,B 0,C 180,E1 -747.111,E2 -747.111} C_VEL
LIN {X 0,Y 601.423,Z 213.572,A -85,B 0,C 180,E1 -749.394,E2 -749.394} C_VEL
LIN {X 0,Y 601.404,Z 213.574,A -85,B 0,C 180,E1 -751.728,E2 -751.728} C_VEL
LIN {X 0,Y 601.427,Z 213.573,A -85,B 0,C 180,E1 -754.119,E2 -754.119} C_VEL
LIN {X 0,Y 601.442,Z 213.569,A -85,B 0,C 180,E1 -757.382,E2 -757.382} C_VEL
LIN {X 0,Y 601.408,Z 213.575,A -85,B 0,C 180,E1 -759.996,E2 -759.996} C_VEL
LIN {X 0,Y 601.42,Z 213.571,A -85,B 0,C 180,E1 -762.67,E2 -762.67} C_VEL
LIN {X 0,Y 601.406,Z 213.574,A -85,B 0,C 180,E1 -765.479,E2 -765.479} C_VEL
LIN {X 0,Y 601.432,Z 213.569,A -85,B 0,C 180,E1 -768.407,E2 -768.407} C_VEL
LIN {X 0,Y 601.414,Z 213.572,A -85,B 0,C 180,E1 -770.873,E2 -770.873} C_VEL
LIN {X 0,Y 601.4,Z 213.575,A -85,B 0,C 180,E1 -773.416,E2 -773.416} C_VEL
LIN {X 0,Y 601.464,Z 213.793,A -85,B 0,C 180,E1 -774.16,E2 -774.16} C_VEL
LIN {X 0,Y 601.553,Z 220.8,A -85,B 0,C 180,E1 -776.37,E2 -776.37} C_VEL
LIN {X 0,Y 601.548,Z 229.698,A -85,B 0,C 180,E1 -779.065,E2 -779.065} C_VEL
LIN {X 0,Y 601.453,Z 239.117,A -85,B 0,C 180,E1 -781.754,E2 -781.754} C_VEL
LIN {X 0,Y 601.476,Z 248.392,A -85,B 0,C 180,E1 -784.384,E2 -784.384} C_VEL
LIN {X 0,Y 601.408,Z 257.659,A -85,B 0,C 180,E1 -786.953,E2 -786.953} C_VEL
LIN {X 0,Y 601.427,Z 266.927,A -85,B 0,C 180,E1 -789.477,E2 -789.477} C_VEL
LIN {X 0,Y 601.405,Z 277.518,A -85,B 0,C 180,E1 -792.311,E2 -792.311} C_VEL
LIN {X 0,Y 601.369,Z 288.109,A -85,B 0,C 180,E1 -795.101,E2 -795.101} C_VEL
LIN {X 0,Y 601.353,Z 298.7,A -85,B 0,C 180,E1 -797.856,E2 -797.856} C_VEL
LIN {X 0,Y 601.381,Z 299.528,A -85,B 0,C 180,E1 -798.07,E2 -798.07} C_VEL
LIN {X 0,Y 601.611,Z 311.239,A -85,B 0,C 180,E1 -798.31,E2 -798.31} C_VEL
LIN {X 0,Y 601.535,Z 324.326,A -85,B 0,C 180,E1 -798.691,E2 -798.691} C_VEL
LIN {X 0,Y 601.484,Z 335.223,A -85,B 0,C 180,E1 -799.131,E2 -799.131} C_VEL
LIN {X 0,Y 601.483,Z 346.746,A -85,B 0,C 180,E1 -799.735,E2 -799.735} C_VEL
LIN {X 0,Y 601.462,Z 358.244,A -85,B 0,C 180,E1 -800.499,E2 -800.499} C_VEL
LIN {X 0,Y 601.436,Z 367.529,A -85,B 0,C 180,E1 -801.262,E2 -801.262} C_VEL
LIN {X 0,Y 601.401,Z 375.984,A -85,B 0,C 180,E1 -802.107,E2 -802.107} C_VEL
LIN {X 0,Y 601.383,Z 384.231,A -85,B 0,C 180,E1 -803.12,E2 -803.12} C_VEL
LIN {X 0,Y 601.373,Z 390.873,A -85,B 0,C 180,E1 -804.13,E2 -804.13} C_VEL
LIN {X 0,Y 601.336,Z 396.947,A -85,B 0,C 180,E1 -805.307,E2 -805.307} C_VEL
LIN {X 0,Y 601.368,Z 400.894,A -85,B 0,C 180,E1 -806.314,E2 -806.314} C_VEL
LIN {X 0,Y 601.325,Z 403.807,A -85,B 0,C 180,E1 -807.32,E2 -807.32} C_VEL
LIN {X 0,Y 601.343,Z 405.201,A -85,B 0,C 180,E1 -807.99,E2 -807.99} C_VEL
LIN {X 0,Y 601.339,Z 406.783,A -85,B 0,C 180,E1 -809.33,E2 -809.33} C_VEL
LIN {X 0,Y 601.335,Z 407,A -85,B 0,C 180,E1 -809.999,E2 -809.999} C_VEL
LIN {X 0,Y 601.347,Z 406.185,A -85,B 0,C 180,E1 -811.339,E2 -811.339} C_VEL
LIN {X 0,Y 601.343,Z 405.203,A -85,B 0,C 180,E1 -812.009,E2 -812.009} C_VEL
LIN {X 0,Y 601.325,Z 403.811,A -85,B 0,C 180,E1 -812.679,E2 -812.679} C_VEL
LIN {X 0,Y 601.368,Z 400.898,A -85,B 0,C 180,E1 -813.685,E2 -813.685} C_VEL
LIN {X 0,Y 601.336,Z 396.953,A -85,B 0,C 180,E1 -814.692,E2 -814.692} C_VEL
LIN {X 0,Y 601.373,Z 390.881,A -85,B 0,C 180,E1 -815.869,E2 -815.869} C_VEL
LIN {X 0,Y 601.381,Z 384.241,A -85,B 0,C 180,E1 -816.879,E2 -816.879} C_VEL
LIN {X 0,Y 601.4,Z 375.996,A -85,B 0,C 180,E1 -817.892,E2 -817.892} C_VEL
LIN {X 0,Y 601.436,Z 367.545,A -85,B 0,C 180,E1 -818.737,E2 -818.737} C_VEL
LIN {X 0,Y 601.451,Z 357.102,A -85,B 0,C 180,E1 -819.584,E2 -819.584} C_VEL
LIN {X 0,Y 601.483,Z 346.769,A -85,B 0,C 180,E1 -820.264,E2 -820.264} C_VEL
LIN {X 0,Y 601.483,Z 335.228,A -85,B 0,C 180,E1 -820.869,E2 -820.869} C_VEL
LIN {X 0,Y 601.526,Z 322.354,A -85,B 0,C 180,E1 -821.375,E2 -821.375} C_VEL
LIN {X 0,Y 601.617,Z 309.468,A -85,B 0,C 180,E1 -821.731,E2 -821.731} C_VEL
LIN {X 0,Y 601.381,Z 299.533,A -85,B 0,C 180,E1 -821.929,E2 -821.929} C_VEL
LIN {X 0,Y 601.385,Z 289.438,A -85,B 0,C 180,E1 -824.551,E2 -824.551} C_VEL
LIN {X 0,Y 601.39,Z 278.847,A -85,B 0,C 180,E1 -827.337,E2 -827.337} C_VEL
LIN {X 0,Y 601.426,Z 268.256,A -85,B 0,C 180,E1 -830.164,E2 -830.164} C_VEL
LIN {X 0,Y 601.408,Z 258.989,A -85,B 0,C 180,E1 -832.682,E2 -832.682} C_VEL
LIN {X 0,Y 601.439,Z 249.721,A -85,B 0,C 180,E1 -835.246,E2 -835.246} C_VEL
LIN {X 0,Y 601.453,Z 239.062,A -85,B 0,C 180,E1 -838.244,E2 -838.244} C_VEL
LIN {X 0,Y 601.479,Z 232.335,A -85,B 0,C 180,E1 -840.16,E2 -840.16} C_VEL
LIN {X 0,Y 601.539,Z 223.682,A -85,B 0,C 180,E1 -842.732,E2 -842.732} C_VEL
LIN {X 0,Y 601.58,Z 216.005,A -85,B 0,C 180,E1 -845.136,E2 -845.136} C_VEL
LIN {X 0,Y 601.409,Z 213.575,A -85,B 0,C 180,E1 -845.977,E2 -845.977} C_VEL
LIN {X 0,Y 601.428,Z 213.572,A -85,B 0,C 180,E1 -848.47,E2 -848.47} C_VEL
LIN {X 0,Y 601.417,Z 213.575,A -85,B 0,C 180,E1 -850.873,E2 -850.873} C_VEL
LIN {X 0,Y 601.449,Z 213.567,A -85,B 0,C 180,E1 -853.583,E2 -853.583} C_VEL
LIN {X 0,Y 601.428,Z 213.572,A -85,B 0,C 180,E1 -856.426,E2 -856.426} C_VEL
LIN {X 0,Y 601.435,Z 213.569,A -85,B 0,C 180,E1 -859.423,E2 -859.423} C_VEL
LIN {X 0,Y 601.419,Z 213.571,A -85,B 0,C 180,E1 -861.731,E2 -861.731} C_VEL
LIN {X 0,Y 601.388,Z 213.576,A -85,B 0,C 180,E1 -864.245,E2 -864.245} C_VEL
LIN {X 0,Y 601.416,Z 213.574,A -85,B 0,C 180,E1 -866.685,E2 -866.685} C_VEL
LIN {X 0,Y 601.402,Z 213.576,A -85,B 0,C 180,E1 -869.056,E2 -869.056} C_VEL
LIN {X 0,Y 601.431,Z 213.572,A -85,B 0,C 180,E1 -871.372,E2 -871.372} C_VEL
LIN {X 0,Y 601.404,Z 213.575,A -85,B 0,C 180,E1 -873.636,E2 -873.636} C_VEL
LIN {X 0,Y 601.457,Z 213.569,A -85,B 0,C 180,E1 -875.859,E2 -875.859} C_VEL
LIN {X 0,Y 601.408,Z 213.572,A -85,B 0,C 180,E1 -878.76,E2 -878.76} C_VEL
LIN {X 0,Y 601.417,Z 213.573,A -85,B 0,C 180,E1 -881.607,E2 -881.607} C_VEL
LIN {X 0,Y 601.416,Z 213.571,A -85,B 0,C 180,E1 -884.408,E2 -884.408} C_VEL
LIN {X 0,Y 601.419,Z 213.574,A -85,B 0,C 180,E1 -887.171,E2 -887.171} C_VEL
LIN {X 0,Y 601.426,Z 213.57,A -85,B 0,C 180,E1 -889.904,E2 -889.904} C_VEL
LIN {X 0,Y 601.452,Z 213.568,A -85,B 0,C 180,E1 -892.614,E2 -892.614} C_VEL
LIN {X 0,Y 601.415,Z 213.573,A -85,B 0,C 180,E1 -895.307,E2 -895.307} C_VEL
LIN {X 0,Y 601.413,Z 213.572,A -85,B 0,C 180,E1 -897.99,E2 -897.99} C_VEL
LIN {X 0,Y 601.458,Z 213.569,A -85,B 0,C 180,E1 -900.668,E2 -900.668} C_VEL
LIN {X 0,Y 601.423,Z 213.571,A -85,B 0,C 180,E1 -903.349,E2 -903.349} C_VEL
LIN {X 0,Y 601.401,Z 213.574,A -85,B 0,C 180,E1 -906.036,E2 -906.036} C_VEL
LIN {X 0,Y 601.437,Z 213.571,A -85,B 0,C 180,E1 -908.736,E2 -908.736} C_VEL
LIN {X 0,Y 601.428,Z 213.57,A -85,B 0,C 180,E1 -911.457,E2 -911.457} C_VEL
LIN {X 0,Y 601.407,Z 213.573,A -85,B 0,C 180,E1 -912.379,E2 -912.379} C_VEL
LIN {X 0,Y 600.744,Z 213.657,A -85,B 0,C 180,E1 -912.938,E2 -912.938} C_VEL
LIN {X 0,Y 597.892,Z 214.011,A -85,B 0,C 180,E1 -913.846,E2 -913.846} C_VEL
LIN {X 0,Y 595.479,Z 214.312,A -85,B 0,C 180,E1 -914.576,E2 -914.576} C_VEL
LIN {X 0,Y 594.442,Z 214.441,A -85,B 0,C 180,E1 -915.14,E2 -915.14} C_VEL
LIN {X 0,Y 594.357,Z 214.45,A -85,B 0,C 180,E1 -915.33,E2 -915.33} C_VEL
LIN {X 0,Y 594.383,Z 214.448,A -85,B 0,C 180,E1 -917.192,E2 -917.192} C_VEL
LIN {X 0,Y 594.315,Z 214.459,A -85,B 0,C 180,E1 -917.905,E2 -917.905} C_VEL
LIN {X 0,Y 594.29,Z 216.829,A -85,B 0,C 180,E1 -920.055,E2 -920.055} C_VEL
LIN {X 0,Y 594.295,Z 220.338,A -85,B 0,C 180,E1 -922.969,E2 -922.969} C_VEL
LIN {X 0,Y 594.277,Z 223.004,A -85,B 0,C 180,E1 -925.196,E2 -925.196} C_VEL
LIN {X 0,Y 594.231,Z 226.479,A -85,B 0,C 180,E1 -928.233,E2 -928.233} C_VEL
LIN {X 0,Y 594.237,Z 229.509,A -85,B 0,C 180,E1 -930.566,E2 -930.566} C_VEL
LIN {X 0,Y 594.232,Z 232.67,A -85,B 0,C 180,E1 -932.958,E2 -932.958} C_VEL
LIN {X 0,Y 594.191,Z 235.974,A -85,B 0,C 180,E1 -935.418,E2 -935.418} C_VEL
LIN {X 0,Y 594.182,Z 239.425,A -85,B 0,C 180,E1 -937.954,E2 -937.954} C_VEL
LIN {X 0,Y 594.198,Z 243.35,A -85,B 0,C 180,E1 -940.803,E2 -940.803} C_VEL
LIN {X 0,Y 594.195,Z 243.679,A -85,B 0,C 180,E1 -941.04,E2 -941.04} C_VEL
LIN {X 0,Y 594.665,Z 249.1,A -85,B 0,C 180,E1 -941.166,E2 -941.166} C_VEL
LIN {X 0,Y 594.582,Z 262.222,A -85,B 0,C 180,E1 -941.531,E2 -941.531} C_VEL
LIN {X 0,Y 594.498,Z 274.285,A -85,B 0,C 180,E1 -942.005,E2 -942.005} C_VEL
LIN {X 0,Y 594.449,Z 286.015,A -85,B 0,C 180,E1 -942.613,E2 -942.613} C_VEL
LIN {X 0,Y 594.462,Z 296.317,A -85,B 0,C 180,E1 -943.289,E2 -943.289} C_VEL
LIN {X 0,Y 594.401,Z 306.488,A -85,B 0,C 180,E1 -944.11,E2 -944.11} C_VEL
LIN {X 0,Y 594.36,Z 315.713,A -85,B 0,C 180,E1 -945.027,E2 -945.027} C_VEL
LIN {X 0,Y 594.314,Z 323.541,A -85,B 0,C 180,E1 -945.987,E2 -945.987} C_VEL
LIN {X 0,Y 594.305,Z 331.15,A -85,B 0,C 180,E1 -947.152,E2 -947.152} C_VEL
LIN {X 0,Y 594.292,Z 336.326,A -85,B 0,C 180,E1 -948.159,E2 -948.159} C_VEL
LIN {X 0,Y 594.245,Z 341.237,A -85,B 0,C 180,E1 -949.424,E2 -949.424} C_VEL
LIN {X 0,Y 594.225,Z 343.747,A -85,B 0,C 180,E1 -950.308,E2 -950.308} C_VEL
LIN {X 0,Y 594.225,Z 345.69,A -85,B 0,C 180,E1 -951.312,E2 -951.312} C_VEL
LIN {X 0,Y 594.239,Z 346.812,A -85,B 0,C 180,E1 -952.408,E2 -952.408} C_VEL
LIN {X 0,Y 594.242,Z 346.766,A -85,B 0,C 180,E1 -953.749,E2 -953.749} C_VEL
LIN {X 0,Y 594.22,Z 345.829,A -85,B 0,C 180,E1 -954.692,E2 -954.692} C_VEL
LIN {X 0,Y 594.242,Z 343.494,A -85,B 0,C 180,E1 -955.878,E2 -955.878} C_VEL
LIN {X 0,Y 594.252,Z 339.712,A -85,B 0,C 180,E1 -957.104,E2 -957.104} C_VEL
LIN {X 0,Y 594.275,Z 335.356,A -85,B 0,C 180,E1 -958.136,E2 -958.136} C_VEL
LIN {X 0,Y 594.302,Z 329.361,A -85,B 0,C 180,E1 -959.24,E2 -959.24} C_VEL
LIN {X 0,Y 594.315,Z 322.682,A -85,B 0,C 180,E1 -960.221,E2 -960.221} C_VEL
LIN {X 0,Y 594.345,Z 314.306,A -85,B 0,C 180,E1 -961.214,E2 -961.214} C_VEL
LIN {X 0,Y 594.401,Z 304.527,A -85,B 0,C 180,E1 -962.153,E2 -962.153} C_VEL
LIN {X 0,Y 594.463,Z 294.608,A -85,B 0,C 180,E1 -962.925,E2 -962.925} C_VEL
LIN {X 0,Y 594.491,Z 282.639,A -85,B 0,C 180,E1 -963.666,E2 -963.666} C_VEL
LIN {X 0,Y 594.538,Z 270.445,A -85,B 0,C 180,E1 -964.252,E2 -964.252} C_VEL
LIN {X 0,Y 594.622,Z 257.705,A -85,B 0,C 180,E1 -964.702,E2 -964.702} C_VEL
LIN {X 0,Y 594.503,Z 245.525,A -85,B 0,C 180,E1 -965,E2 -965} C_VEL
LIN {X 0,Y 594.266,Z 243.662,A -85,B 0,C 180,E1 -965.06,E2 -965.06} C_VEL
LIN {X 0,Y 594.254,Z 239.933,A -85,B 0,C 180,E1 -967.763,E2 -967.763} C_VEL
LIN {X 0,Y 594.215,Z 236.962,A -85,B 0,C 180,E1 -969.941,E2 -969.941} C_VEL
LIN {X 0,Y 594.214,Z 234.062,A -85,B 0,C 180,E1 -972.091,E2 -972.091} C_VEL
LIN {X 0,Y 594.245,Z 231.23,A -85,B 0,C 180,E1 -974.217,E2 -974.217} C_VEL
LIN {X 0,Y 594.234,Z 227.566,A -85,B 0,C 180,E1 -977.015,E2 -977.015} C_VEL
LIN {X 0,Y 594.254,Z 224.987,A -85,B 0,C 180,E1 -979.093,E2 -979.093} C_VEL
LIN {X 0,Y 594.283,Z 221.7,A -85,B 0,C 180,E1 -981.842,E2 -981.842} C_VEL
LIN {X 0,Y 594.275,Z 219.245,A -85,B 0,C 180,E1 -983.891,E2 -983.891} C_VEL
LIN {X 0,Y 594.276,Z 215.958,A -85,B 0,C 180,E1 -986.611,E2 -986.611} C_VEL
LIN {X 0,Y 594.332,Z 214.457,A -85,B 0,C 180,E1 -987.968,E2 -987.968} C_VEL
LIN {X 0,Y 594.398,Z 214.445,A -85,B 0,C 180,E1 -990.001,E2 -990.001} C_VEL
LIN {X 0,Y 594.399,Z 214.447,A -85,B 0,C 180,E1 -992.711,E2 -992.711} C_VEL
LIN {X 0,Y 594.39,Z 214.448,A -85,B 0,C 180,E1 -995.428,E2 -995.428} C_VEL
LIN {X 0,Y 594.406,Z 214.444,A -85,B 0,C 180,E1 -998.157,E2 -998.157} C_VEL
LIN {X 0,Y 594.383,Z 214.449,A -85,B 0,C 180,E1 -1001.079,E2 -1001.079} C_VEL
LIN {X 0,Y 594.377,Z 214.448,A -85,B 0,C 180,E1 -1003.68,E2 -1003.68} C_VEL
LIN {X 0,Y 594.385,Z 214.45,A -85,B 0,C 180,E1 -1006.722,E2 -1006.722} C_VEL
LIN {X 0,Y 594.359,Z 214.45,A -85,B 0,C 180,E1 -1009.335,E2 -1009.335} C_VEL
LIN {X 0,Y 594.36,Z 214.451,A -85,B 0,C 180,E1 -1011.504,E2 -1011.504} C_VEL
LIN {X 0,Y 594.381,Z 214.449,A -85,B 0,C 180,E1 -1013.705,E2 -1013.705} C_VEL
LIN {X 0,Y 594.383,Z 214.449,A -85,B 0,C 180,E1 -1016.7,E2 -1016.7} C_VEL
LIN {X 0,Y 594.377,Z 214.449,A -85,B 0,C 180,E1 -1018.999,E2 -1018.999} C_VEL
LIN {X 0,Y 594.386,Z 214.449,A -85,B 0,C 180,E1 -1021.647,E2 -1021.647} C_VEL
LIN {X 0,Y 594.393,Z 214.447,A -85,B 0,C 180,E1 -1024.58,E2 -1024.58} C_VEL
LIN {X 0,Y 594.381,Z 214.45,A -85,B 0,C 180,E1 -1027.088,E2 -1027.088} C_VEL
LIN {X 0,Y 594.371,Z 214.45,A -85,B 0,C 180,E1 -1029.776,E2 -1029.776} C_VEL
LIN {X 0,Y 594.384,Z 214.447,A -85,B 0,C 180,E1 -1032.375,E2 -1032.375} C_VEL
LIN {X 0,Y 594.358,Z 214.454,A -85,B 0,C 180,E1 -1035.193,E2 -1035.193} C_VEL
LIN {X 0,Y 594.383,Z 214.447,A -85,B 0,C 180,E1 -1038.153,E2 -1038.153} C_VEL
LIN {X 0,Y 594.385,Z 214.448,A -85,B 0,C 180,E1 -1041.197,E2 -1041.197} C_VEL
LIN {X 0,Y 594.394,Z 214.446,A -85,B 0,C 180,E1 -1043.76,E2 -1043.76} C_VEL
LIN {X 0,Y 594.381,Z 214.448,A -85,B 0,C 180,E1 -1046.241,E2 -1046.241} C_VEL
LIN {X 0,Y 594.369,Z 214.45,A -85,B 0,C 180,E1 -1048.651,E2 -1048.651} C_VEL
LIN {X 0,Y 594.384,Z 214.449,A -85,B 0,C 180,E1 -1051.043,E2 -1051.043} C_VEL
LIN {X 0,Y 594.388,Z 214.447,A -85,B 0,C 180,E1 -1053.978,E2 -1053.978} C_VEL
LIN {X 0,Y 594.378,Z 214.448,A -85,B 0,C 180,E1 -1056.297,E2 -1056.297} C_VEL
LIN {X 0,Y 594.408,Z 214.447,A -85,B 0,C 180,E1 -1059.226,E2 -1059.226} C_VEL
LIN {X 0,Y 594.356,Z 214.451,A -85,B 0,C 180,E1 -1062.096,E2 -1062.096} C_VEL
LIN {X 0,Y 594.364,Z 214.45,A -85,B 0,C 180,E1 -1064.22,E2 -1064.22} C_VEL
LIN {X 0,Y 594.381,Z 214.449,A -85,B 0,C 180,E1 -1066.322,E2 -1066.322} C_VEL
LIN {X 0,Y 594.375,Z 214.448,A -85,B 0,C 180,E1 -1069.096,E2 -1069.096} C_VEL
LIN {X 0,Y 594.385,Z 214.451,A -85,B 0,C 180,E1 -1071.844,E2 -1071.844} C_VEL
LIN {X 0,Y 594.385,Z 214.447,A -85,B 0,C 180,E1 -1074.573,E2 -1074.573} C_VEL
LIN {X 0,Y 594.409,Z 214.445,A -85,B 0,C 180,E1 -1077.29,E2 -1077.29} C_VEL
LIN {X 0,Y 594.416,Z 214.445,A -85,B 0,C 180,E1 -1080.001,E2 -1080.001} C_VEL
LIN {X 0,Y 594.4,Z 214.445,A -85,B 0,C 180,E1 -1082.712,E2 -1082.712} C_VEL
LIN {X 0,Y 594.393,Z 214.448,A -85,B 0,C 180,E1 -1085.429,E2 -1085.429} C_VEL
LIN {X 0,Y 594.387,Z 214.448,A -85,B 0,C 180,E1 -1088.158,E2 -1088.158} C_VEL
LIN {X 0,Y 594.388,Z 214.448,A -85,B 0,C 180,E1 -1091.069,E2 -1091.069} C_VEL
LIN {X 0,Y 594.377,Z 214.451,A -85,B 0,C 180,E1 -1093.68,E2 -1093.68} C_VEL
LIN {X 0,Y 594.394,Z 214.446,A -85,B 0,C 180,E1 -1096.486,E2 -1096.486} C_VEL
LIN {X 0,Y 594.371,Z 214.452,A -85,B 0,C 180,E1 -1099.335,E2 -1099.335} C_VEL
LIN {X 0,Y 594.367,Z 214.452,A -85,B 0,C 180,E1 -1101.504,E2 -1101.504} C_VEL
LIN {X 0,Y 594.375,Z 214.448,A -85,B 0,C 180,E1 -1104.447,E2 -1104.447} C_VEL
LIN {X 0,Y 594.39,Z 214.446,A -85,B 0,C 180,E1 -1106.7,E2 -1106.7} C_VEL
LIN {X 0,Y 594.39,Z 214.446,A -85,B 0,C 180,E1 -1108.999,E2 -1108.999} C_VEL
LIN {X 0,Y 594.382,Z 214.448,A -85,B 0,C 180,E1 -1111.642,E2 -1111.642} C_VEL
LIN {X 0,Y 594.385,Z 214.447,A -85,B 0,C 180,E1 -1114.58,E2 -1114.58} C_VEL
LIN {X 0,Y 594.394,Z 214.449,A -85,B 0,C 180,E1 -1117.608,E2 -1117.608} C_VEL
LIN {X 0,Y 594.373,Z 214.449,A -85,B 0,C 180,E1 -1120.567,E2 -1120.567} C_VEL
LIN {X 0,Y 594.375,Z 214.451,A -85,B 0,C 180,E1 -1123.3,E2 -1123.3} C_VEL
LIN {X 0,Y 594.368,Z 214.449,A -85,B 0,C 180,E1 -1126.161,E2 -1126.161} C_VEL
LIN {X 0,Y 594.389,Z 214.446,A -85,B 0,C 180,E1 -1128.536,E2 -1128.536} C_VEL
LIN {X 0,Y 594.378,Z 214.451,A -85,B 0,C 180,E1 -1131.297,E2 -1131.297} C_VEL
LIN {X 0,Y 594.393,Z 214.564,A -85,B 0,C 180,E1 -1133.915,E2 -1133.915} C_VEL
LIN {X 0,Y 594.617,Z 219.223,A -85,B 0,C 180,E1 -1135.435,E2 -1135.435} C_VEL
LIN {X 0,Y 594.554,Z 227.046,A -85,B 0,C 180,E1 -1137.863,E2 -1137.863} C_VEL
LIN {X 0,Y 594.482,Z 234.983,A -85,B 0,C 180,E1 -1140.229,E2 -1140.229} C_VEL
LIN {X 0,Y 594.439,Z 244.411,A -85,B 0,C 180,E1 -1142.923,E2 -1142.923} C_VEL
LIN {X 0,Y 594.443,Z 253.688,A -85,B 0,C 180,E1 -1145.556,E2 -1145.556} C_VEL
LIN {X 0,Y 594.39,Z 264.279,A -85,B 0,C 180,E1 -1148.497,E2 -1148.497} C_VEL
LIN {X 0,Y 594.38,Z 274.87,A -85,B 0,C 180,E1 -1151.382,E2 -1151.382} C_VEL
LIN {X 0,Y 594.326,Z 285.461,A -85,B 0,C 180,E1 -1154.217,E2 -1154.217} C_VEL
LIN {X 0,Y 594.318,Z 294.729,A -85,B 0,C 180,E1 -1156.667,E2 -1156.667} C_VEL
LIN {X 0,Y 594.293,Z 299.528,A -85,B 0,C 180,E1 -1157.926,E2 -1157.926} C_VEL
LIN {X 0,Y 594.676,Z 305.194,A -85,B 0,C 180,E1 -1158.042,E2 -1158.042} C_VEL
LIN {X 0,Y 594.617,Z 318.473,A -85,B 0,C 180,E1 -1158.365,E2 -1158.365} C_VEL
LIN {X 0,Y 594.533,Z 330.622,A -85,B 0,C 180,E1 -1158.8,E2 -1158.8} C_VEL
LIN {X 0,Y 594.479,Z 342.198,A -85,B 0,C 180,E1 -1159.354,E2 -1159.354} C_VEL
LIN {X 0,Y 594.471,Z 353.467,A -85,B 0,C 180,E1 -1160.043,E2 -1160.043} C_VEL
LIN {X 0,Y 594.406,Z 363.639,A -85,B 0,C 180,E1 -1160.815,E2 -1160.815} C_VEL
LIN {X 0,Y 594.373,Z 372.781,A -85,B 0,C 180,E1 -1161.671,E2 -1161.671} C_VEL
LIN {X 0,Y 594.317,Z 381.685,A -85,B 0,C 180,E1 -1162.696,E2 -1162.696} C_VEL
LIN {X 0,Y 594.281,Z 388.171,A -85,B 0,C 180,E1 -1163.615,E2 -1163.615} C_VEL
LIN {X 0,Y 594.289,Z 393.677,A -85,B 0,C 180,E1 -1164.571,E2 -1164.571} C_VEL
LIN {X 0,Y 594.27,Z 398.368,A -85,B 0,C 180,E1 -1165.591,E2 -1165.591} C_VEL
LIN {X 0,Y 594.267,Z 401.954,A -85,B 0,C 180,E1 -1166.609,E2 -1166.609} C_VEL
LIN {X 0,Y 594.226,Z 403.807,A -85,B 0,C 180,E1 -1167.288,E2 -1167.288} C_VEL
LIN {X 0,Y 594.242,Z 405.2,A -85,B 0,C 180,E1 -1167.966,E2 -1167.966} C_VEL
LIN {X 0,Y 594.239,Z 406.784,A -85,B 0,C 180,E1 -1169.322,E2 -1169.322} C_VEL
LIN {X 0,Y 594.236,Z 407,A -85,B 0,C 180,E1 -1169.999,E2 -1169.999} C_VEL
LIN {X 0,Y 594.247,Z 406.186,A -85,B 0,C 180,E1 -1171.355,E2 -1171.355} C_VEL
LIN {X 0,Y 594.242,Z 405.203,A -85,B 0,C 180,E1 -1172.033,E2 -1172.033} C_VEL
LIN {X 0,Y 594.226,Z 403.811,A -85,B 0,C 180,E1 -1172.711,E2 -1172.711} C_VEL
LIN {X 0,Y 594.289,Z 400.898,A -85,B 0,C 180,E1 -1173.729,E2 -1173.729} C_VEL
LIN {X 0,Y 594.241,Z 396.952,A -85,B 0,C 180,E1 -1174.748,E2 -1174.748} C_VEL
LIN {X 0,Y 594.305,Z 390.882,A -85,B 0,C 180,E1 -1175.939,E2 -1175.939} C_VEL
LIN {X 0,Y 594.308,Z 384.241,A -85,B 0,C 180,E1 -1176.961,E2 -1176.961} C_VEL
LIN {X 0,Y 594.359,Z 375.996,A -85,B 0,C 180,E1 -1177.986,E2 -1177.986} C_VEL
LIN {X 0,Y 594.382,Z 367.545,A -85,B 0,C 180,E1 -1178.841,E2 -1178.841} C_VEL
LIN {X 0,Y 594.435,Z 357.103,A -85,B 0,C 180,E1 -1179.699,E2 -1179.699} C_VEL
LIN {X 0,Y 594.458,Z 346.771,A -85,B 0,C 180,E1 -1180.386,E2 -1180.386} C_VEL
LIN {X 0,Y 594.501,Z 334.784,A -85,B 0,C 180,E1 -1181.018,E2 -1181.018} C_VEL
LIN {X 0,Y 594.563,Z 322.51,A -85,B 0,C 180,E1 -1181.505,E2 -1181.505} C_VEL
LIN {X 0,Y 594.678,Z 309.467,A -85,B 0,C 180,E1 -1181.87,E2 -1181.87} C_VEL
LIN {X 0,Y 594.447,Z 300.724,A -85,B 0,C 180,E1 -1182.04,E2 -1182.04} C_VEL
LIN {X 0,Y 594.292,Z 299.533,A -85,B 0,C 180,E1 -1182.073,E2 -1182.073} C_VEL
LIN {X 0,Y 594.313,Z 289.438,A -85,B 0,C 180,E1 -1184.728,E2 -1184.728} C_VEL
LIN {X 0,Y 594.336,Z 278.847,A -85,B 0,C 180,E1 -1187.549,E2 -1187.549} C_VEL
LIN {X 0,Y 594.39,Z 269.58,A -85,B 0,C 180,E1 -1190.052,E2 -1190.052} C_VEL
LIN {X 0,Y 594.374,Z 259.816,A -85,B 0,C 180,E1 -1192.736,E2 -1192.736} C_VEL
LIN {X 0,Y 594.427,Z 251.045,A -85,B 0,C 180,E1 -1195.19,E2 -1195.19} C_VEL
LIN {X 0,Y 594.454,Z 241.504,A -85,B 0,C 180,E1 -1197.843,E2 -1197.843} C_VEL
LIN {X 0,Y 594.488,Z 232.948,A -85,B 0,C 180,E1 -1200.344,E2 -1200.344} C_VEL
LIN {X 0,Y 594.561,Z 224.38,A -85,B 0,C 180,E1 -1202.938,E2 -1202.938} C_VEL
LIN {X 0,Y 594.6,Z 216.69,A -85,B 0,C 180,E1 -1205.391,E2 -1205.391} C_VEL
LIN {X 0,Y 594.355,Z 214.454,A -85,B 0,C 180,E1 -1206.191,E2 -1206.191} C_VEL
LIN {X 0,Y 594.386,Z 214.449,A -85,B 0,C 180,E1 -1208.804,E2 -1208.804} C_VEL
LIN {X 0,Y 594.386,Z 214.449,A -85,B 0,C 180,E1 -1211.848,E2 -1211.848} C_VEL
LIN {X 0,Y 594.381,Z 214.451,A -85,B 0,C 180,E1 -1214.235,E2 -1214.235} C_VEL
LIN {X 0,Y 594.365,Z 214.45,A -85,B 0,C 180,E1 -1217.147,E2 -1217.147} C_VEL
LIN {X 0,Y 594.389,Z 214.447,A -85,B 0,C 180,E1 -1219.434,E2 -1219.434} C_VEL
LIN {X 0,Y 594.388,Z 214.449,A -85,B 0,C 180,E1 -1222.391,E2 -1222.391} C_VEL
LIN {X 0,Y 594.396,Z 214.447,A -85,B 0,C 180,E1 -1225.42,E2 -1225.42} C_VEL
LIN {X 0,Y 594.374,Z 214.449,A -85,B 0,C 180,E1 -1228.356,E2 -1228.356} C_VEL
LIN {X 0,Y 594.382,Z 214.449,A -85,B 0,C 180,E1 -1231.041,E2 -1231.041} C_VEL
LIN {X 0,Y 594.381,Z 214.448,A -85,B 0,C 180,E1 -1233.977,E2 -1233.977} C_VEL
LIN {X 0,Y 594.375,Z 214.448,A -85,B 0,C 180,E1 -1236.295,E2 -1236.295} C_VEL
LIN {X 0,Y 594.402,Z 214.448,A -85,B 0,C 180,E1 -1239.224,E2 -1239.224} C_VEL
LIN {X 0,Y 594.352,Z 214.451,A -85,B 0,C 180,E1 -1242.094,E2 -1242.094} C_VEL
LIN {X 0,Y 594.368,Z 214.449,A -85,B 0,C 180,E1 -1244.218,E2 -1244.218} C_VEL
LIN {X 0,Y 594.368,Z 214.451,A -85,B 0,C 180,E1 -1247.016,E2 -1247.016} C_VEL
LIN {X 0,Y 594.387,Z 214.447,A -85,B 0,C 180,E1 -1249.783,E2 -1249.783} C_VEL
LIN {X 0,Y 594.4,Z 214.446,A -85,B 0,C 180,E1 -1252.526,E2 -1252.526} C_VEL
LIN {X 0,Y 594.386,Z 214.449,A -85,B 0,C 180,E1 -1255.251,E2 -1255.251} C_VEL
LIN {X 0,Y 594.385,Z 214.447,A -85,B 0,C 180,E1 -1257.966,E2 -1257.966} C_VEL
LIN {X 0,Y 594.427,Z 214.445,A -85,B 0,C 180,E1 -1260.676,E2 -1260.676} C_VEL
LIN {X 0,Y 594.375,Z 214.449,A -85,B 0,C 180,E1 -1263.388,E2 -1263.388} C_VEL
LIN {X 0,Y 594.358,Z 214.451,A -85,B 0,C 180,E1 -1266.108,E2 -1266.108} C_VEL
LIN {X 0,Y 594.397,Z 214.447,A -85,B 0,C 180,E1 -1268.841,E2 -1268.841} C_VEL
LIN {X 0,Y 594.387,Z 214.447,A -85,B 0,C 180,E1 -1271.595,E2 -1271.595} C_VEL
LIN {X 0,Y 594.381,Z 214.451,A -85,B 0,C 180,E1 -1274.376,E2 -1274.376} C_VEL
LIN {X 0,Y 594.357,Z 214.45,A -85,B 0,C 180,E1 -1275.33,E2 -1275.33} C_VEL
LIN {X 0,Y 593.683,Z 214.554,A -85,B 0,C 180,E1 -1275.897,E2 -1275.897} C_VEL
LIN {X 0,Y 590.798,Z 214.896,A -85,B 0,C 180,E1 -1276.815,E2 -1276.815} C_VEL
LIN {X 0,Y 588.362,Z 215.2,A -85,B 0,C 180,E1 -1277.554,E2 -1277.554} C_VEL
LIN {X 0,Y 587.315,Z 215.38,A -85,B 0,C 180,E1 -1278.123,E2 -1278.123} C_VEL
LIN {X 0,Y 587.229,Z 215.519,A -85,B 0,C 180,E1 -1278.315,E2 -1278.315} C_VEL
LIN {X 0,Y 587.23,Z 218.641,A -85,B 0,C 180,E1 -1281.04,E2 -1281.04} C_VEL
LIN {X 0,Y 587.231,Z 221.301,A -85,B 0,C 180,E1 -1283.261,E2 -1283.261} C_VEL
LIN {X 0,Y 587.201,Z 224.799,A -85,B 0,C 180,E1 -1286.151,E2 -1286.151} C_VEL
LIN {X 0,Y 587.146,Z 227.999,A -85,B 0,C 180,E1 -1289.099,E2 -1289.099} C_VEL
LIN {X 0,Y 587.116,Z 231.488,A -85,B 0,C 180,E1 -1291.801,E2 -1291.801} C_VEL
LIN {X 0,Y 587.109,Z 234.798,A -85,B 0,C 180,E1 -1294.315,E2 -1294.315} C_VEL
LIN {X 0,Y 587.094,Z 238.071,A -85,B 0,C 180,E1 -1296.764,E2 -1296.764} C_VEL
LIN {X 0,Y 587.092,Z 241.609,A -85,B 0,C 180,E1 -1299.378,E2 -1299.378} C_VEL
LIN {X 0,Y 587.108,Z 243.682,A -85,B 0,C 180,E1 -1300.896,E2 -1300.896} C_VEL
LIN {X 0,Y 587.714,Z 249.084,A -85,B 0,C 180,E1 -1301.023,E2 -1301.023} C_VEL
LIN {X 0,Y 587.638,Z 261.147,A -85,B 0,C 180,E1 -1301.357,E2 -1301.357} C_VEL
LIN {X 0,Y 587.525,Z 273.226,A -85,B 0,C 180,E1 -1301.825,E2 -1301.825} C_VEL
LIN {X 0,Y 587.467,Z 284.695,A -85,B 0,C 180,E1 -1302.41,E2 -1302.41} C_VEL
LIN {X 0,Y 587.453,Z 295.812,A -85,B 0,C 180,E1 -1303.134,E2 -1303.134} C_VEL
LIN {X 0,Y 587.359,Z 305.849,A -85,B 0,C 180,E1 -1303.945,E2 -1303.945} C_VEL
LIN {X 0,Y 587.292,Z 315.552,A -85,B 0,C 180,E1 -1304.911,E2 -1304.911} C_VEL
LIN {X 0,Y 587.24,Z 323.48,A -85,B 0,C 180,E1 -1305.893,E2 -1305.893} C_VEL
LIN {X 0,Y 587.211,Z 330.594,A -85,B 0,C 180,E1 -1306.985,E2 -1306.985} C_VEL
LIN {X 0,Y 587.197,Z 336.539,A -85,B 0,C 180,E1 -1308.145,E2 -1308.145} C_VEL
LIN {X 0,Y 587.156,Z 341.106,A -85,B 0,C 180,E1 -1309.338,E2 -1309.338} C_VEL
LIN {X 0,Y 587.128,Z 344.5,A -85,B 0,C 180,E1 -1310.624,E2 -1310.624} C_VEL
LIN {X 0,Y 587.123,Z 345.992,A -85,B 0,C 180,E1 -1311.506,E2 -1311.506} C_VEL
LIN {X 0,Y 587.154,Z 346.798,A -85,B 0,C 180,E1 -1312.379,E2 -1312.379} C_VEL
LIN {X 0,Y 587.123,Z 346.944,A -85,B 0,C 180,E1 -1313.319,E2 -1313.319} C_VEL
LIN {X 0,Y 587.131,Z 346.111,A -85,B 0,C 180,E1 -1314.482,E2 -1314.482} C_VEL
LIN {X 0,Y 587.139,Z 343.863,A -85,B 0,C 180,E1 -1315.766,E2 -1315.766} C_VEL
LIN {X 0,Y 587.147,Z 340.574,A -85,B 0,C 180,E1 -1316.914,E2 -1316.914} C_VEL
LIN {X 0,Y 587.201,Z 335.418,A -85,B 0,C 180,E1 -1318.184,E2 -1318.184} C_VEL
LIN {X 0,Y 587.234,Z 329.474,A -85,B 0,C 180,E1 -1319.295,E2 -1319.295} C_VEL
LIN {X 0,Y 587.267,Z 321.819,A -85,B 0,C 180,E1 -1320.42,E2 -1320.42} C_VEL
LIN {X 0,Y 587.305,Z 313.458,A -85,B 0,C 180,E1 -1321.403,E2 -1321.403} C_VEL
LIN {X 0,Y 587.371,Z 304.111,A -85,B 0,C 180,E1 -1322.3,E2 -1322.3} C_VEL
LIN {X 0,Y 587.434,Z 294.448,A -85,B 0,C 180,E1 -1323.056,E2 -1323.056} C_VEL
LIN {X 0,Y 587.488,Z 282.721,A -85,B 0,C 180,E1 -1323.79,E2 -1323.79} C_VEL
LIN {X 0,Y 587.566,Z 270.15,A -85,B 0,C 180,E1 -1324.4,E2 -1324.4} C_VEL
LIN {X 0,Y 587.688,Z 257.202,A -85,B 0,C 180,E1 -1324.856,E2 -1324.856} C_VEL
LIN {X 0,Y 587.513,Z 246.22,A -85,B 0,C 180,E1 -1325.132,E2 -1325.132} C_VEL
LIN {X 0,Y 587.161,Z 243.742,A -85,B 0,C 180,E1 -1325.186,E2 -1325.186} C_VEL
LIN {X 0,Y 587.133,Z 239.563,A -85,B 0,C 180,E1 -1328.219,E2 -1328.219} C_VEL
LIN {X 0,Y 587.175,Z 235.632,A -85,B 0,C 180,E1 -1331.146,E2 -1331.146} C_VEL
LIN {X 0,Y 587.161,Z 231.836,A -85,B 0,C 180,E1 -1334.021,E2 -1334.021} C_VEL
LIN {X 0,Y 587.161,Z 228.163,A -85,B 0,C 180,E1 -1336.856,E2 -1336.856} C_VEL
LIN {X 0,Y 587.169,Z 224.944,A -85,B 0,C 180,E1 -1339.658,E2 -1339.658} C_VEL
LIN {X 0,Y 587.219,Z 222.392,A -85,B 0,C 180,E1 -1341.743,E2 -1341.743} C_VEL
LIN {X 0,Y 587.227,Z 219.916,A -85,B 0,C 180,E1 -1343.817,E2 -1343.817} C_VEL
LIN {X 0,Y 587.201,Z 216.622,A -85,B 0,C 180,E1 -1346.57,E2 -1346.57} C_VEL
LIN {X 0,Y 587.304,Z 215.332,A -85,B 0,C 180,E1 -1347.943,E2 -1347.943} C_VEL
LIN {X 0,Y 587.367,Z 215.321,A -85,B 0,C 180,E1 -1350.001,E2 -1350.001} C_VEL
LIN {X 0,Y 587.364,Z 215.323,A -85,B 0,C 180,E1 -1352.744,E2 -1352.744} C_VEL
LIN {X 0,Y 587.354,Z 215.324,A -85,B 0,C 180,E1 -1355.494,E2 -1355.494} C_VEL
LIN {X 0,Y 587.36,Z 215.322,A -85,B 0,C 180,E1 -1358.256,E2 -1358.256} C_VEL
LIN {X 0,Y 587.348,Z 215.325,A -85,B 0,C 180,E1 -1361.142,E2 -1361.142} C_VEL
LIN {X 0,Y 587.352,Z 215.326,A -85,B 0,C 180,E1 -1364.262,E2 -1364.262} C_VEL
LIN {X 0,Y 587.349,Z 215.324,A -85,B 0,C 180,E1 -1367.407,E2 -1367.407} C_VEL
LIN {X 0,Y 587.327,Z 215.327,A -85,B 0,C 180,E1 -1370.306,E2 -1370.306} C_VEL
LIN {X 0,Y 587.356,Z 215.324,A -85,B 0,C 180,E1 -1373.258,E2 -1373.258} C_VEL
LIN {X 0,Y 587.356,Z 215.323,A -85,B 0,C 180,E1 -1376.278,E2 -1376.278} C_VEL
LIN {X 0,Y 587.344,Z 215.327,A -85,B 0,C 180,E1 -1379.136,E2 -1379.136} C_VEL
LIN {X 0,Y 587.351,Z 215.324,A -85,B 0,C 180,E1 -1381.84,E2 -1381.84} C_VEL
LIN {X 0,Y 587.352,Z 215.323,A -85,B 0,C 180,E1 -1384.351,E2 -1384.351} C_VEL
LIN {X 0,Y 587.346,Z 215.324,A -85,B 0,C 180,E1 -1386.748,E2 -1386.748} C_VEL
LIN {X 0,Y 587.339,Z 215.327,A -85,B 0,C 180,E1 -1389.361,E2 -1389.361} C_VEL
LIN {X 0,Y 587.332,Z 215.326,A -85,B 0,C 180,E1 -1392.11,E2 -1392.11} C_VEL
LIN {X 0,Y 587.31,Z 215.33,A -85,B 0,C 180,E1 -1395.09,E2 -1395.09} C_VEL
LIN {X 0,Y 587.348,Z 215.324,A -85,B 0,C 180,E1 -1397.929,E2 -1397.929} C_VEL
LIN {X 0,Y 587.333,Z 215.328,A -85,B 0,C 180,E1 -1401.059,E2 -1401.059} C_VEL
LIN {X 0,Y 587.351,Z 215.326,A -85,B 0,C 180,E1 -1403.293,E2 -1403.293} C_VEL
LIN {X 0,Y 587.36,Z 215.323,A -85,B 0,C 180,E1 -1405.782,E2 -1405.782} C_VEL
LIN {X 0,Y 587.34,Z 215.325,A -85,B 0,C 180,E1 -1408.233,E2 -1408.233} C_VEL
LIN {X 0,Y 587.35,Z 215.324,A -85,B 0,C 180,E1 -1410.868,E2 -1410.868} C_VEL
LIN {X 0,Y 587.36,Z 215.323,A -85,B 0,C 180,E1 -1413.82,E2 -1413.82} C_VEL
LIN {X 0,Y 587.331,Z 215.328,A -85,B 0,C 180,E1 -1415.995,E2 -1415.995} C_VEL
LIN {X 0,Y 587.322,Z 215.329,A -85,B 0,C 180,E1 -1418.227,E2 -1418.227} C_VEL
LIN {X 0,Y 587.35,Z 215.323,A -85,B 0,C 180,E1 -1421.153,E2 -1421.153} C_VEL
LIN {X 0,Y 587.32,Z 215.329,A -85,B 0,C 180,E1 -1424.026,E2 -1424.026} C_VEL
LIN {X 0,Y 587.361,Z 215.325,A -85,B 0,C 180,E1 -1426.156,E2 -1426.156} C_VEL
LIN {X 0,Y 587.342,Z 215.324,A -85,B 0,C 180,E1 -1428.964,E2 -1428.964} C_VEL
LIN {X 0,Y 587.345,Z 215.326,A -85,B 0,C 180,E1 -1431.746,E2 -1431.746} C_VEL
LIN {X 0,Y 587.353,Z 215.323,A -85,B 0,C 180,E1 -1434.508,E2 -1434.508} C_VEL
LIN {X 0,Y 587.375,Z 215.321,A -85,B 0,C 180,E1 -1437.258,E2 -1437.258} C_VEL
LIN {X 0,Y 587.386,Z 215.321,A -85,B 0,C 180,E1 -1440.001,E2 -1440.001} C_VEL
LIN {X 0,Y 587.368,Z 215.321,A -85,B 0,C 180,E1 -1442.744,E2 -1442.744} C_VEL
LIN {X 0,Y 587.357,Z 215.325,A -85,B 0,C 180,E1 -1445.494,E2 -1445.494} C_VEL
LIN {X 0,Y 587.347,Z 215.324,A -85,B 0,C 180,E1 -1448.256,E2 -1448.256} C_VEL
LIN {X 0,Y 587.357,Z 215.324,A -85,B 0,C 180,E1 -1451.134,E2 -1451.134} C_VEL
LIN {X 0,Y 587.356,Z 215.324,A -85,B 0,C 180,E1 -1453.847,E2 -1453.847} C_VEL
LIN {X 0,Y 587.344,Z 215.325,A -85,B 0,C 180,E1 -1456.81,E2 -1456.81} C_VEL
LIN {X 0,Y 587.318,Z 215.328,A -85,B 0,C 180,E1 -1459.577,E2 -1459.577} C_VEL
LIN {X 0,Y 587.323,Z 215.328,A -85,B 0,C 180,E1 -1461.775,E2 -1461.775} C_VEL
LIN {X 0,Y 587.318,Z 215.328,A -85,B 0,C 180,E1 -1464.761,E2 -1464.761} C_VEL
LIN {X 0,Y 587.337,Z 215.326,A -85,B 0,C 180,E1 -1467.047,E2 -1467.047} C_VEL
LIN {X 0,Y 587.35,Z 215.325,A -85,B 0,C 180,E1 -1469.38,E2 -1469.38} C_VEL
LIN {X 0,Y 587.348,Z 215.326,A -85,B 0,C 180,E1 -1471.835,E2 -1471.835} C_VEL
LIN {X 0,Y 587.35,Z 215.325,A -85,B 0,C 180,E1 -1474.347,E2 -1474.347} C_VEL
LIN {X 0,Y 587.349,Z 215.327,A -85,B 0,C 180,E1 -1477.608,E2 -1477.608} C_VEL
LIN {X 0,Y 587.318,Z 215.328,A -85,B 0,C 180,E1 -1480.255,E2 -1480.255} C_VEL
LIN {X 0,Y 587.324,Z 215.328,A -85,B 0,C 180,E1 -1483.118,E2 -1483.118} C_VEL
LIN {X 0,Y 587.32,Z 215.327,A -85,B 0,C 180,E1 -1486.048,E2 -1486.048} C_VEL
LIN {X 0,Y 587.343,Z 215.326,A -85,B 0,C 180,E1 -1488.925,E2 -1488.925} C_VEL
LIN {X 0,Y 587.326,Z 215.329,A -85,B 0,C 180,E1 -1491.52,E2 -1491.52} C_VEL
LIN {X 0,Y 587.348,Z 215.386,A -85,B 0,C 180,E1 -1493.679,E2 -1493.679} C_VEL
LIN {X 0,Y 587.665,Z 219.221,A -85,B 0,C 180,E1 -1494.967,E2 -1494.967} C_VEL
LIN {X 0,Y 587.585,Z 228.242,A -85,B 0,C 180,E1 -1497.822,E2 -1497.822} C_VEL
LIN {X 0,Y 587.489,Z 236.212,A -85,B 0,C 180,E1 -1500.234,E2 -1500.234} C_VEL
LIN {X 0,Y 587.42,Z 245.661,A -85,B 0,C 180,E1 -1502.958,E2 -1502.958} C_VEL
LIN {X 0,Y 587.417,Z 254.262,A -85,B 0,C 180,E1 -1505.407,E2 -1505.407} C_VEL
LIN {X 0,Y 587.389,Z 264.279,A -85,B 0,C 180,E1 -1508.228,E2 -1508.228} C_VEL
LIN {X 0,Y 587.313,Z 274.87,A -85,B 0,C 180,E1 -1511.149,E2 -1511.149} C_VEL
LIN {X 0,Y 587.263,Z 285.461,A -85,B 0,C 180,E1 -1514.022,E2 -1514.022} C_VEL
LIN {X 0,Y 587.229,Z 296.052,A -85,B 0,C 180,E1 -1516.856,E2 -1516.856} C_VEL
LIN {X 0,Y 587.204,Z 299.528,A -85,B 0,C 180,E1 -1517.778,E2 -1517.778} C_VEL
LIN {X 0,Y 587.731,Z 305.194,A -85,B 0,C 180,E1 -1517.898,E2 -1517.898} C_VEL
LIN {X 0,Y 587.685,Z 318.474,A -85,B 0,C 180,E1 -1518.226,E2 -1518.226} C_VEL
LIN {X 0,Y 587.566,Z 330.404,A -85,B 0,C 180,E1 -1518.656,E2 -1518.656} C_VEL
LIN {X 0,Y 587.479,Z 342.199,A -85,B 0,C 180,E1 -1519.226,E2 -1519.226} C_VEL
LIN {X 0,Y 587.467,Z 353.469,A -85,B 0,C 180,E1 -1519.923,E2 -1519.923} C_VEL
LIN {X 0,Y 587.385,Z 363.639,A -85,B 0,C 180,E1 -1520.704,E2 -1520.704} C_VEL
LIN {X 0,Y 587.331,Z 372.781,A -85,B 0,C 180,E1 -1521.57,E2 -1521.57} C_VEL
LIN {X 0,Y 587.26,Z 381.685,A -85,B 0,C 180,E1 -1522.608,E2 -1522.608} C_VEL
LIN {X 0,Y 587.195,Z 388.748,A -85,B 0,C 180,E1 -1523.627,E2 -1523.627} C_VEL
LIN {X 0,Y 587.212,Z 393.677,A -85,B 0,C 180,E1 -1524.505,E2 -1524.505} C_VEL
LIN {X 0,Y 587.189,Z 398.369,A -85,B 0,C 180,E1 -1525.537,E2 -1525.537} C_VEL
LIN {X 0,Y 587.194,Z 401.954,A -85,B 0,C 180,E1 -1526.568,E2 -1526.568} C_VEL
LIN {X 0,Y 587.132,Z 403.807,A -85,B 0,C 180,E1 -1527.255,E2 -1527.255} C_VEL
LIN {X 0,Y 587.141,Z 405.199,A -85,B 0,C 180,E1 -1527.941,E2 -1527.941} C_VEL
LIN {X 0,Y 587.14,Z 406.784,A -85,B 0,C 180,E1 -1529.313,E2 -1529.313} C_VEL
LIN {X 0,Y 587.137,Z 407,A -85,B 0,C 180,E1 -1529.999,E2 -1529.999} C_VEL
LIN {X 0,Y 587.147,Z 406.186,A -85,B 0,C 180,E1 -1531.371,E2 -1531.371} C_VEL
LIN {X 0,Y 587.141,Z 405.202,A -85,B 0,C 180,E1 -1532.057,E2 -1532.057} C_VEL
LIN {X 0,Y 587.132,Z 403.811,A -85,B 0,C 180,E1 -1532.744,E2 -1532.744} C_VEL
LIN {X 0,Y 587.213,Z 400.898,A -85,B 0,C 180,E1 -1533.774,E2 -1533.774} C_VEL
LIN {X 0,Y 587.147,Z 396.952,A -85,B 0,C 180,E1 -1534.806,E2 -1534.806} C_VEL
LIN {X 0,Y 587.218,Z 390.881,A -85,B 0,C 180,E1 -1536.01,E2 -1536.01} C_VEL
LIN {X 0,Y 587.245,Z 384.242,A -85,B 0,C 180,E1 -1537.045,E2 -1537.045} C_VEL
LIN {X 0,Y 587.299,Z 375.996,A -85,B 0,C 180,E1 -1538.082,E2 -1538.082} C_VEL
LIN {X 0,Y 587.343,Z 367.546,A -85,B 0,C 180,E1 -1538.948,E2 -1538.948} C_VEL
LIN {X 0,Y 587.421,Z 357.105,A -85,B 0,C 180,E1 -1539.816,E2 -1539.816} C_VEL
LIN {X 0,Y 587.475,Z 346.769,A -85,B 0,C 180,E1 -1540.511,E2 -1540.511} C_VEL
LIN {X 0,Y 587.53,Z 335.171,A -85,B 0,C 180,E1 -1541.133,E2 -1541.133} C_VEL
LIN {X 0,Y 587.624,Z 322.712,A -85,B 0,C 180,E1 -1541.636,E2 -1541.636} C_VEL
LIN {X 0,Y 587.713,Z 309.466,A -85,B 0,C 180,E1 -1542.013,E2 -1542.013} C_VEL
LIN {X 0,Y 587.507,Z 301.662,A -85,B 0,C 180,E1 -1542.171,E2 -1542.171} C_VEL
LIN {X 0,Y 587.203,Z 299.533,A -85,B 0,C 180,E1 -1542.221,E2 -1542.221} C_VEL
LIN {X 0,Y 587.259,Z 289.438,A -85,B 0,C 180,E1 -1544.909,E2 -1544.909} C_VEL
LIN {X 0,Y 587.303,Z 278.847,A -85,B 0,C 180,E1 -1547.766,E2 -1547.766} C_VEL
LIN {X 0,Y 587.37,Z 268.256,A -85,B 0,C 180,E1 -1550.668,E2 -1550.668} C_VEL
LIN {X 0,Y 587.388,Z 258.989,A -85,B 0,C 180,E1 -1553.255,E2 -1553.255} C_VEL
LIN {X 0,Y 587.449,Z 249.742,A -85,B 0,C 180,E1 -1555.85,E2 -1555.85} C_VEL
LIN {X 0,Y 587.417,Z 241.285,A -85,B 0,C 180,E1 -1558.202,E2 -1558.202} C_VEL
LIN {X 0,Y 587.556,Z 232.177,A -85,B 0,C 180,E1 -1560.952,E2 -1560.952} C_VEL
LIN {X 0,Y 587.645,Z 223.063,A -85,B 0,C 180,E1 -1563.787,E2 -1563.787} C_VEL
LIN {X 0,Y 587.575,Z 216.712,A -85,B 0,C 180,E1 -1565.879,E2 -1565.879} C_VEL
LIN {X 0,Y 587.321,Z 215.33,A -85,B 0,C 180,E1 -1566.418,E2 -1566.418} C_VEL
LIN {X 0,Y 587.346,Z 215.325,A -85,B 0,C 180,E1 -1569.358,E2 -1569.358} C_VEL
LIN {X 0,Y 587.334,Z 215.328,A -85,B 0,C 180,E1 -1572.107,E2 -1572.107} C_VEL
LIN {X 0,Y 587.304,Z 215.33,A -85,B 0,C 180,E1 -1574.911,E2 -1574.911} C_VEL
LIN {X 0,Y 587.352,Z 215.324,A -85,B 0,C 180,E1 -1577.927,E2 -1577.927} C_VEL
LIN {X 0,Y 587.332,Z 215.326,A -85,B 0,C 180,E1 -1580.639,E2 -1580.639} C_VEL
LIN {X 0,Y 587.346,Z 215.327,A -85,B 0,C 180,E1 -1583.291,E2 -1583.291} C_VEL
LIN {X 0,Y 587.365,Z 215.323,A -85,B 0,C 180,E1 -1585.779,E2 -1585.779} C_VEL
LIN {X 0,Y 587.338,Z 215.325,A -85,B 0,C 180,E1 -1588.23,E2 -1588.23} C_VEL
LIN {X 0,Y 587.349,Z 215.324,A -85,B 0,C 180,E1 -1590.865,E2 -1590.865} C_VEL
LIN {X 0,Y 587.356,Z 215.324,A -85,B 0,C 180,E1 -1593.818,E2 -1593.818} C_VEL
LIN {X 0,Y 587.327,Z 215.328,A -85,B 0,C 180,E1 -1595.992,E2 -1595.992} C_VEL
LIN {X 0,Y 587.318,Z 215.329,A -85,B 0,C 180,E1 -1598.225,E2 -1598.225} C_VEL
LIN {X 0,Y 587.351,Z 215.324,A -85,B 0,C 180,E1 -1601.15,E2 -1601.15} C_VEL
LIN {X 0,Y 587.326,Z 215.327,A -85,B 0,C 180,E1 -1604.024,E2 -1604.024} C_VEL
LIN {X 0,Y 587.36,Z 215.324,A -85,B 0,C 180,E1 -1606.153,E2 -1606.153} C_VEL
LIN {X 0,Y 587.341,Z 215.325,A -85,B 0,C 180,E1 -1608.962,E2 -1608.962} C_VEL
LIN {X 0,Y 587.366,Z 215.324,A -85,B 0,C 180,E1 -1611.744,E2 -1611.744} C_VEL
LIN {X 0,Y 587.362,Z 215.322,A -85,B 0,C 180,E1 -1614.506,E2 -1614.506} C_VEL
LIN {X 0,Y 587.375,Z 215.323,A -85,B 0,C 180,E1 -1617.256,E2 -1617.256} C_VEL
LIN {X 0,Y 587.378,Z 215.32,A -85,B 0,C 180,E1 -1619.999,E2 -1619.999} C_VEL
LIN {X 0,Y 587.376,Z 215.321,A -85,B 0,C 180,E1 -1622.742,E2 -1622.742} C_VEL
LIN {X 0,Y 587.358,Z 215.324,A -85,B 0,C 180,E1 -1625.492,E2 -1625.492} C_VEL
LIN {X 0,Y 587.368,Z 215.322,A -85,B 0,C 180,E1 -1628.254,E2 -1628.254} C_VEL
LIN {X 0,Y 587.355,Z 215.324,A -85,B 0,C 180,E1 -1631.14,E2 -1631.14} C_VEL
LIN {X 0,Y 587.356,Z 215.326,A -85,B 0,C 180,E1 -1634.26,E2 -1634.26} C_VEL
LIN {X 0,Y 587.334,Z 215.327,A -85,B 0,C 180,E1 -1637.405,E2 -1637.405} C_VEL
LIN {X 0,Y 587.229,Z 215.519,A -85,B 0,C 180,E1 -1638.315,E2 -1638.315} C_VEL
LIN {X 0,Y 586.568,Z 216.162,A -85,B 0,C 180,E1 -1638.884,E2 -1638.884} C_VEL
LIN {X 0,Y 583.734,Z 217.482,A -85,B 0,C 180,E1 -1639.804,E2 -1639.804} C_VEL
LIN {X 0,Y 581.322,Z 218.599,A -85,B 0,C 180,E1 -1640.543,E2 -1640.543} C_VEL
LIN {X 0,Y 580.261,Z 219.366,A -85,B 0,C 180,E1 -1641.114,E2 -1641.114} C_VEL
LIN {X 0,Y 580.162,Z 219.603,A -85,B 0,C 180,E1 -1641.308,E2 -1641.308} C_VEL
LIN {X 0,Y 580.154,Z 222.268,A -85,B 0,C 180,E1 -1643.562,E2 -1643.562} C_VEL
LIN {X 0,Y 580.126,Z 225.582,A -85,B 0,C 180,E1 -1646.303,E2 -1646.303} C_VEL
LIN {X 0,Y 580.089,Z 228.567,A -85,B 0,C 180,E1 -1648.986,E2 -1648.986} C_VEL
LIN {X 0,Y 580.027,Z 231.321,A -85,B 0,C 180,E1 -1651.399,E2 -1651.399} C_VEL
LIN {X 0,Y 580.027,Z 234.529,A -85,B 0,C 180,E1 -1653.872,E2 -1653.872} C_VEL
LIN {X 0,Y 579.99,Z 237.89,A -85,B 0,C 180,E1 -1656.422,E2 -1656.422} C_VEL
LIN {X 0,Y 580.002,Z 241.533,A -85,B 0,C 180,E1 -1659.151,E2 -1659.151} C_VEL
LIN {X 0,Y 580.03,Z 243.686,A -85,B 0,C 180,E1 -1660.748,E2 -1660.748} C_VEL
LIN {X 0,Y 580.768,Z 249.811,A -85,B 0,C 180,E1 -1660.894,E2 -1660.894} C_VEL
LIN {X 0,Y 580.685,Z 261.968,A -85,B 0,C 180,E1 -1661.243,E2 -1661.243} C_VEL
LIN {X 0,Y 580.56,Z 274.42,A -85,B 0,C 180,E1 -1661.742,E2 -1661.742} C_VEL
LIN {X 0,Y 580.485,Z 285.439,A -85,B 0,C 180,E1 -1662.324,E2 -1662.324} C_VEL
LIN {X 0,Y 580.438,Z 296.234,A -85,B 0,C 180,E1 -1663.045,E2 -1663.045} C_VEL
LIN {X 0,Y 580.325,Z 306.488,A -85,B 0,C 180,E1 -1663.892,E2 -1663.892} C_VEL
LIN {X 0,Y 580.255,Z 315.029,A -85,B 0,C 180,E1 -1664.754,E2 -1664.754} C_VEL
LIN {X 0,Y 580.186,Z 323.388,A -85,B 0,C 180,E1 -1665.793,E2 -1665.793} C_VEL
LIN {X 0,Y 580.124,Z 330.819,A -85,B 0,C 180,E1 -1666.95,E2 -1666.95} C_VEL
LIN {X 0,Y 580.106,Z 335.823,A -85,B 0,C 180,E1 -1667.931,E2 -1667.931} C_VEL
LIN {X 0,Y 580.082,Z 340.611,A -85,B 0,C 180,E1 -1669.139,E2 -1669.139} C_VEL
LIN {X 0,Y 580.076,Z 343.261,A -85,B 0,C 180,E1 -1670.05,E2 -1670.05} C_VEL
LIN {X 0,Y 580.049,Z 345.177,A -85,B 0,C 180,E1 -1670.948,E2 -1670.948} C_VEL
LIN {X 0,Y 580.032,Z 346.514,A -85,B 0,C 180,E1 -1671.957,E2 -1671.957} C_VEL
LIN {X 0,Y 580.031,Z 346.994,A -85,B 0,C 180,E1 -1673.098,E2 -1673.098} C_VEL
LIN {X 0,Y 580.041,Z 346.18,A -85,B 0,C 180,E1 -1674.439,E2 -1674.439} C_VEL
LIN {X 0,Y 580.043,Z 344.541,A -85,B 0,C 180,E1 -1675.475,E2 -1675.475} C_VEL
LIN {X 0,Y 580.064,Z 341.352,A -85,B 0,C 180,E1 -1676.717,E2 -1676.717} C_VEL
LIN {X 0,Y 580.09,Z 336.563,A -85,B 0,C 180,E1 -1678,E2 -1678} C_VEL
LIN {X 0,Y 580.133,Z 331.662,A -85,B 0,C 180,E1 -1678.993,E2 -1678.993} C_VEL
LIN {X 0,Y 580.16,Z 325.342,A -85,B 0,C 180,E1 -1680.021,E2 -1680.021} C_VEL
LIN {X 0,Y 580.242,Z 317.731,A -85,B 0,C 180,E1 -1681.022,E2 -1681.022} C_VEL
LIN {X 0,Y 580.299,Z 308.52,A -85,B 0,C 180,E1 -1682.008,E2 -1682.008} C_VEL
LIN {X 0,Y 580.402,Z 298.2,A -85,B 0,C 180,E1 -1682.898,E2 -1682.898} C_VEL
LIN {X 0,Y 580.506,Z 286.504,A -85,B 0,C 180,E1 -1683.7,E2 -1683.7} C_VEL
LIN {X 0,Y 580.599,Z 276.17,A -85,B 0,C 180,E1 -1684.263,E2 -1684.263} C_VEL
LIN {X 0,Y 580.662,Z 264.879,A -85,B 0,C 180,E1 -1684.746,E2 -1684.746} C_VEL
LIN {X 0,Y 580.757,Z 251.769,A -85,B 0,C 180,E1 -1685.148,E2 -1685.148} C_VEL
LIN {X 0,Y 580.522,Z 246.69,A -85,B 0,C 180,E1 -1685.27,E2 -1685.27} C_VEL
LIN {X 0,Y 580.076,Z 243.67,A -85,B 0,C 180,E1 -1685.353,E2 -1685.353} C_VEL
LIN {X 0,Y 580.035,Z 240.192,A -85,B 0,C 180,E1 -1687.939,E2 -1687.939} C_VEL
LIN {X 0,Y 580.052,Z 237.223,A -85,B 0,C 180,E1 -1690.169,E2 -1690.169} C_VEL
LIN {X 0,Y 580.058,Z 233.295,A -85,B 0,C 180,E1 -1693.163,E2 -1693.163} C_VEL
LIN {X 0,Y 580.112,Z 229.748,A -85,B 0,C 180,E1 -1695.979,E2 -1695.979} C_VEL
LIN {X 0,Y 580.14,Z 226.435,A -85,B 0,C 180,E1 -1698.881,E2 -1698.881} C_VEL
LIN {X 0,Y 580.164,Z 223.083,A -85,B 0,C 180,E1 -1701.642,E2 -1701.642} C_VEL
LIN {X 0,Y 580.179,Z 220.596,A -85,B 0,C 180,E1 -1703.742,E2 -1703.742} C_VEL
LIN {X 0,Y 580.129,Z 217.296,A -85,B 0,C 180,E1 -1706.528,E2 -1706.528} C_VEL
LIN {X 0,Y 580.135,Z 216.487,A -85,B 0,C 180,E1 -1707.223,E2 -1707.223} C_VEL
LIN {X 0,Y 580.282,Z 216.205,A -85,B 0,C 180,E1 -1708.613,E2 -1708.613} C_VEL
LIN {X 0,Y 580.36,Z 216.197,A -85,B 0,C 180,E1 -1710.695,E2 -1710.695} C_VEL
LIN {X 0,Y 580.277,Z 216.204,A -85,B 0,C 180,E1 -1713.472,E2 -1713.472} C_VEL
LIN {X 0,Y 580.318,Z 216.2,A -85,B 0,C 180,E1 -1715.56,E2 -1715.56} C_VEL
LIN {X 0,Y 580.324,Z 216.199,A -85,B 0,C 180,E1 -1718.357,E2 -1718.357} C_VEL
LIN {X 0,Y 580.319,Z 216.2,A -85,B 0,C 180,E1 -1721.209,E2 -1721.209} C_VEL
LIN {X 0,Y 580.316,Z 216.2,A -85,B 0,C 180,E1 -1724.018,E2 -1724.018} C_VEL
LIN {X 0,Y 580.301,Z 216.202,A -85,B 0,C 180,E1 -1726.916,E2 -1726.916} C_VEL
LIN {X 0,Y 580.298,Z 216.203,A -85,B 0,C 180,E1 -1729.823,E2 -1729.823} C_VEL
LIN {X 0,Y 580.318,Z 216.2,A -85,B 0,C 180,E1 -1732.802,E2 -1732.802} C_VEL
LIN {X 0,Y 580.299,Z 216.202,A -85,B 0,C 180,E1 -1735.081,E2 -1735.081} C_VEL
LIN {X 0,Y 580.311,Z 216.202,A -85,B 0,C 180,E1 -1737.865,E2 -1737.865} C_VEL
LIN {X 0,Y 580.283,Z 216.204,A -85,B 0,C 180,E1 -1740.698,E2 -1740.698} C_VEL
LIN {X 0,Y 580.297,Z 216.202,A -85,B 0,C 180,E1 -1743.318,E2 -1743.318} C_VEL
LIN {X 0,Y 580.319,Z 216.2,A -85,B 0,C 180,E1 -1745.769,E2 -1745.769} C_VEL
LIN {X 0,Y 580.281,Z 216.205,A -85,B 0,C 180,E1 -1748.148,E2 -1748.148} C_VEL
LIN {X 0,Y 580.297,Z 216.203,A -85,B 0,C 180,E1 -1750.844,E2 -1750.844} C_VEL
LIN {X 0,Y 580.285,Z 216.203,A -85,B 0,C 180,E1 -1753.658,E2 -1753.658} C_VEL
LIN {X 0,Y 580.271,Z 216.206,A -85,B 0,C 180,E1 -1756.611,E2 -1756.611} C_VEL
LIN {X 0,Y 580.297,Z 216.202,A -85,B 0,C 180,E1 -1759.159,E2 -1759.159} C_VEL
LIN {X 0,Y 580.287,Z 216.204,A -85,B 0,C 180,E1 -1761.928,E2 -1761.928} C_VEL
LIN {X 0,Y 580.284,Z 216.206,A -85,B 0,C 180,E1 -1764.457,E2 -1764.457} C_VEL
LIN {X 0,Y 580.289,Z 216.203,A -85,B 0,C 180,E1 -1766.977,E2 -1766.977} C_VEL
LIN {X 0,Y 580.295,Z 216.202,A -85,B 0,C 180,E1 -1769.427,E2 -1769.427} C_VEL
LIN {X 0,Y 580.298,Z 216.203,A -85,B 0,C 180,E1 -1772.143,E2 -1772.143} C_VEL
LIN {X 0,Y 580.322,Z 216.198,A -85,B 0,C 180,E1 -1775.271,E2 -1775.271} C_VEL
LIN {X 0,Y 580.273,Z 216.207,A -85,B 0,C 180,E1 -1777.949,E2 -1777.949} C_VEL
LIN {X 0,Y 580.302,Z 216.201,A -85,B 0,C 180,E1 -1780.915,E2 -1780.915} C_VEL
LIN {X 0,Y 580.271,Z 216.208,A -85,B 0,C 180,E1 -1783.827,E2 -1783.827} C_VEL
LIN {X 0,Y 580.328,Z 216.2,A -85,B 0,C 180,E1 -1785.984,E2 -1785.984} C_VEL
LIN {X 0,Y 580.31,Z 216.2,A -85,B 0,C 180,E1 -1788.828,E2 -1788.828} C_VEL
LIN {X 0,Y 580.315,Z 216.201,A -85,B 0,C 180,E1 -1791.645,E2 -1791.645} C_VEL
LIN {X 0,Y 580.291,Z 216.203,A -85,B 0,C 180,E1 -1793.743,E2 -1793.743} C_VEL
LIN {X 0,Y 580.272,Z 216.205,A -85,B 0,C 180,E1 -1795.834,E2 -1795.834} C_VEL
LIN {X 0,Y 580.331,Z 216.198,A -85,B 0,C 180,E1 -1797.919,E2 -1797.919} C_VEL
LIN {X 0,Y 580.358,Z 216.195,A -85,B 0,C 180,E1 -1800.695,E2 -1800.695} C_VEL
LIN {X 0,Y 580.285,Z 216.205,A -85,B 0,C 180,E1 -1803.473,E2 -1803.473} C_VEL
LIN {X 0,Y 580.323,Z 216.202,A -85,B 0,C 180,E1 -1805.561,E2 -1805.561} C_VEL
LIN {X 0,Y 580.331,Z 216.199,A -85,B 0,C 180,E1 -1807.656,E2 -1807.656} C_VEL
LIN {X 0,Y 580.3,Z 216.202,A -85,B 0,C 180,E1 -1810.468,E2 -1810.468} C_VEL
LIN {X 0,Y 580.275,Z 216.205,A -85,B 0,C 180,E1 -1813.305,E2 -1813.305} C_VEL
LIN {X 0,Y 580.298,Z 216.202,A -85,B 0,C 180,E1 -1815.454,E2 -1815.454} C_VEL
LIN {X 0,Y 580.276,Z 216.205,A -85,B 0,C 180,E1 -1817.626,E2 -1817.626} C_VEL
LIN {X 0,Y 580.294,Z 216.202,A -85,B 0,C 180,E1 -1819.824,E2 -1819.824} C_VEL
LIN {X 0,Y 580.275,Z 216.205,A -85,B 0,C 180,E1 -1822.053,E2 -1822.053} C_VEL
LIN {X 0,Y 580.291,Z 216.206,A -85,B 0,C 180,E1 -1825.081,E2 -1825.081} C_VEL
LIN {X 0,Y 580.301,Z 216.201,A -85,B 0,C 180,E1 -1827.858,E2 -1827.858} C_VEL
LIN {X 0,Y 580.281,Z 216.206,A -85,B 0,C 180,E1 -1830.693,E2 -1830.693} C_VEL
LIN {X 0,Y 580.29,Z 216.204,A -85,B 0,C 180,E1 -1833.313,E2 -1833.313} C_VEL
LIN {X 0,Y 580.252,Z 216.207,A -85,B 0,C 180,E1 -1835.756,E2 -1835.756} C_VEL
LIN {X 0,Y 580.291,Z 216.202,A -85,B 0,C 180,E1 -1838.147,E2 -1838.147} C_VEL
LIN {X 0,Y 580.304,Z 216.202,A -85,B 0,C 180,E1 -1840.844,E2 -1840.844} C_VEL
LIN {X 0,Y 580.281,Z 216.205,A -85,B 0,C 180,E1 -1843.658,E2 -1843.658} C_VEL
LIN {X 0,Y 580.281,Z 216.205,A -85,B 0,C 180,E1 -1846.61,E2 -1846.61} C_VEL
LIN {X 0,Y 580.304,Z 216.204,A -85,B 0,C 180,E1 -1849.156,E2 -1849.156} C_VEL
LIN {X 0,Y 580.293,Z 216.203,A -85,B 0,C 180,E1 -1851.928,E2 -1851.928} C_VEL
LIN {X 0,Y 580.328,Z 216.395,A -85,B 0,C 180,E1 -1853.505,E2 -1853.505} C_VEL
LIN {X 0,Y 580.713,Z 220.513,A -85,B 0,C 180,E1 -1854.909,E2 -1854.909} C_VEL
LIN {X 0,Y 580.66,Z 228.272,A -85,B 0,C 180,E1 -1857.411,E2 -1857.411} C_VEL
LIN {X 0,Y 580.492,Z 236.088,A -85,B 0,C 180,E1 -1859.838,E2 -1859.838} C_VEL
LIN {X 0,Y 580.441,Z 245.541,A -85,B 0,C 180,E1 -1862.605,E2 -1862.605} C_VEL
LIN {X 0,Y 580.402,Z 254.787,A -85,B 0,C 180,E1 -1865.254,E2 -1865.254} C_VEL
LIN {X 0,Y 580.361,Z 265.603,A -85,B 0,C 180,E1 -1868.324,E2 -1868.324} C_VEL
LIN {X 0,Y 580.279,Z 276.194,A -85,B 0,C 180,E1 -1871.279,E2 -1871.279} C_VEL
LIN {X 0,Y 580.218,Z 286.785,A -85,B 0,C 180,E1 -1874.184,E2 -1874.184} C_VEL
LIN {X 0,Y 580.178,Z 296.052,A -85,B 0,C 180,E1 -1876.693,E2 -1876.693} C_VEL
LIN {X 0,Y 580.129,Z 299.528,A -85,B 0,C 180,E1 -1877.626,E2 -1877.626} C_VEL
LIN {X 0,Y 580.807,Z 305.194,A -85,B 0,C 180,E1 -1877.752,E2 -1877.752} C_VEL
LIN {X 0,Y 580.721,Z 318.475,A -85,B 0,C 180,E1 -1878.082,E2 -1878.082} C_VEL
LIN {X 0,Y 580.6,Z 330.616,A -85,B 0,C 180,E1 -1878.528,E2 -1878.528} C_VEL
LIN {X 0,Y 580.49,Z 342.198,A -85,B 0,C 180,E1 -1879.095,E2 -1879.095} C_VEL
LIN {X 0,Y 580.456,Z 353.47,A -85,B 0,C 180,E1 -1879.8,E2 -1879.8} C_VEL
LIN {X 0,Y 580.353,Z 363.639,A -85,B 0,C 180,E1 -1880.59,E2 -1880.59} C_VEL
LIN {X 0,Y 580.27,Z 372.78,A -85,B 0,C 180,E1 -1881.467,E2 -1881.467} C_VEL
LIN {X 0,Y 580.2,Z 381.685,A -85,B 0,C 180,E1 -1882.517,E2 -1882.517} C_VEL
LIN {X 0,Y 580.12,Z 388.467,A -85,B 0,C 180,E1 -1883.505,E2 -1883.505} C_VEL
LIN {X 0,Y 580.14,Z 393.676,A -85,B 0,C 180,E1 -1884.438,E2 -1884.438} C_VEL
LIN {X 0,Y 580.108,Z 398.369,A -85,B 0,C 180,E1 -1885.483,E2 -1885.483} C_VEL
LIN {X 0,Y 580.123,Z 401.955,A -85,B 0,C 180,E1 -1886.527,E2 -1886.527} C_VEL
LIN {X 0,Y 580.043,Z 403.807,A -85,B 0,C 180,E1 -1887.221,E2 -1887.221} C_VEL
LIN {X 0,Y 580.04,Z 405.198,A -85,B 0,C 180,E1 -1887.916,E2 -1887.916} C_VEL
LIN {X 0,Y 580.04,Z 406.784,A -85,B 0,C 180,E1 -1889.305,E2 -1889.305} C_VEL
LIN {X 0,Y 580.037,Z 407,A -85,B 0,C 180,E1 -1889.999,E2 -1889.999} C_VEL
LIN {X 0,Y 580.047,Z 406.187,A -85,B 0,C 180,E1 -1891.388,E2 -1891.388} C_VEL
LIN {X 0,Y 580.04,Z 405.201,A -85,B 0,C 180,E1 -1892.082,E2 -1892.082} C_VEL
LIN {X 0,Y 580.043,Z 403.811,A -85,B 0,C 180,E1 -1892.777,E2 -1892.777} C_VEL
LIN {X 0,Y 580.11,Z 400.898,A -85,B 0,C 180,E1 -1893.82,E2 -1893.82} C_VEL
LIN {X 0,Y 580.053,Z 396.952,A -85,B 0,C 180,E1 -1894.865,E2 -1894.865} C_VEL
LIN {X 0,Y 580.139,Z 390.881,A -85,B 0,C 180,E1 -1896.084,E2 -1896.084} C_VEL
LIN {X 0,Y 580.184,Z 384.242,A -85,B 0,C 180,E1 -1897.132,E2 -1897.132} C_VEL
LIN {X 0,Y 580.25,Z 375.996,A -85,B 0,C 180,E1 -1898.181,E2 -1898.181} C_VEL
LIN {X 0,Y 580.308,Z 367.546,A -85,B 0,C 180,E1 -1899.058,E2 -1899.058} C_VEL
LIN {X 0,Y 580.422,Z 357.107,A -85,B 0,C 180,E1 -1899.935,E2 -1899.935} C_VEL
LIN {X 0,Y 580.477,Z 346.768,A -85,B 0,C 180,E1 -1900.639,E2 -1900.639} C_VEL
LIN {X 0,Y 580.563,Z 335.605,A -85,B 0,C 180,E1 -1901.247,E2 -1901.247} C_VEL
LIN {X 0,Y 580.662,Z 323.789,A -85,B 0,C 180,E1 -1901.74,E2 -1901.74} C_VEL
LIN {X 0,Y 580.802,Z 310.379,A -85,B 0,C 180,E1 -1902.136,E2 -1902.136} C_VEL
LIN {X 0,Y 580.602,Z 302.375,A -85,B 0,C 180,E1 -1902.307,E2 -1902.307} C_VEL
LIN {X 0,Y 580.128,Z 299.533,A -85,B 0,C 180,E1 -1902.372,E2 -1902.372} C_VEL
LIN {X 0,Y 580.218,Z 289.438,A -85,B 0,C 180,E1 -1905.094,E2 -1905.094} C_VEL
LIN {X 0,Y 580.255,Z 278.847,A -85,B 0,C 180,E1 -1907.989,E2 -1907.989} C_VEL
LIN {X 0,Y 580.331,Z 268.494,A -85,B 0,C 180,E1 -1910.864,E2 -1910.864} C_VEL
LIN {X 0,Y 580.382,Z 258.989,A -85,B 0,C 180,E1 -1913.553,E2 -1913.553} C_VEL
LIN {X 0,Y 580.387,Z 248.798,A -85,B 0,C 180,E1 -1916.352,E2 -1916.352} C_VEL
LIN {X 0,Y 580.433,Z 239.907,A -85,B 0,C 180,E1 -1918.968,E2 -1918.968} C_VEL
LIN {X 0,Y 580.592,Z 230.955,A -85,B 0,C 180,E1 -1921.719,E2 -1921.719} C_VEL
LIN {X 0,Y 580.707,Z 221.771,A -85,B 0,C 180,E1 -1924.667,E2 -1924.667} C_VEL
LIN {X 0,Y 580.658,Z 218.371,A -85,B 0,C 180,E1 -1925.812,E2 -1925.812} C_VEL
LIN {X 0,Y 580.307,Z 216.204,A -85,B 0,C 180,E1 -1926.59,E2 -1926.59} C_VEL
LIN {X 0,Y 580.308,Z 216.201,A -85,B 0,C 180,E1 -1929.186,E2 -1929.186} C_VEL
LIN {X 0,Y 580.314,Z 216.201,A -85,B 0,C 180,E1 -1931.765,E2 -1931.765} C_VEL
LIN {X 0,Y 580.262,Z 216.207,A -85,B 0,C 180,E1 -1934.625,E2 -1934.625} C_VEL
LIN {X 0,Y 580.286,Z 216.206,A -85,B 0,C 180,E1 -1937.627,E2 -1937.627} C_VEL
LIN {X 0,Y 580.288,Z 216.205,A -85,B 0,C 180,E1 -1940.066,E2 -1940.066} C_VEL
LIN {X 0,Y 580.297,Z 216.203,A -85,B 0,C 180,E1 -1943.065,E2 -1943.065} C_VEL
LIN {X 0,Y 580.317,Z 216.2,A -85,B 0,C 180,E1 -1946.145,E2 -1946.145} C_VEL
LIN {X 0,Y 580.272,Z 216.205,A -85,B 0,C 180,E1 -1948.613,E2 -1948.613} C_VEL
LIN {X 0,Y 580.292,Z 216.204,A -85,B 0,C 180,E1 -1951.023,E2 -1951.023} C_VEL
LIN {X 0,Y 580.29,Z 216.205,A -85,B 0,C 180,E1 -1953.665,E2 -1953.665} C_VEL
LIN {X 0,Y 580.295,Z 216.204,A -85,B 0,C 180,E1 -1955.683,E2 -1955.683} C_VEL
LIN {X 0,Y 580.282,Z 216.204,A -85,B 0,C 180,E1 -1958.694,E2 -1958.694} C_VEL
LIN {X 0,Y 580.316,Z 216.2,A -85,B 0,C 180,E1 -1960.913,E2 -1960.913} C_VEL
LIN {X 0,Y 580.279,Z 216.207,A -85,B 0,C 180,E1 -1963.825,E2 -1963.825} C_VEL
LIN {X 0,Y 580.325,Z 216.202,A -85,B 0,C 180,E1 -1965.982,E2 -1965.982} C_VEL
LIN {X 0,Y 580.3,Z 216.201,A -85,B 0,C 180,E1 -1968.826,E2 -1968.826} C_VEL
LIN {X 0,Y 580.33,Z 216.201,A -85,B 0,C 180,E1 -1971.643,E2 -1971.643} C_VEL
LIN {X 0,Y 580.327,Z 216.198,A -85,B 0,C 180,E1 -1974.439,E2 -1974.439} C_VEL
LIN {X 0,Y 580.341,Z 216.199,A -85,B 0,C 180,E1 -1977.222,E2 -1977.222} C_VEL
LIN {X 0,Y 580.348,Z 216.196,A -85,B 0,C 180,E1 -1979.999,E2 -1979.999} C_VEL
LIN {X 0,Y 580.342,Z 216.198,A -85,B 0,C 180,E1 -1982.775,E2 -1982.775} C_VEL
LIN {X 0,Y 580.322,Z 216.2,A -85,B 0,C 180,E1 -1985.559,E2 -1985.559} C_VEL
LIN {X 0,Y 580.331,Z 216.199,A -85,B 0,C 180,E1 -1988.355,E2 -1988.355} C_VEL
LIN {X 0,Y 580.326,Z 216.199,A -85,B 0,C 180,E1 -1991.207,E2 -1991.207} C_VEL
LIN {X 0,Y 580.307,Z 216.204,A -85,B 0,C 180,E1 -1994.338,E2 -1994.338} C_VEL
LIN {X 0,Y 580.305,Z 216.202,A -85,B 0,C 180,E1 -1996.914,E2 -1996.914} C_VEL
LIN {X 0,Y 580.16,Z 216.222,A -85,B 0,C 180,E1 -1998.357,E2 -1998.357} C_VEL
LIN {X 0,Y 580.183,Z 219.4,A -85,B 0,C 180,E1 -2001.137,E2 -2001.137} C_VEL
LIN {X 0,Y 580.162,Z 219.603,A -85,B 0,C 180,E1 -2001.308,E2 -2001.308} C_VEL
LIN {X 0,Y 579.454,Z 220.347,A -85,B 0,C 180,E1 -2001.883,E2 -2001.883} C_VEL
LIN {X 0,Y 576.565,Z 221.709,A -85,B 0,C 180,E1 -2002.814,E2 -2002.814} C_VEL
LIN {X 0,Y 574.158,Z 222.802,A -85,B 0,C 180,E1 -2003.563,E2 -2003.563} C_VEL
LIN {X 0,Y 573.141,Z 223.572,A -85,B 0,C 180,E1 -2004.142,E2 -2004.142} C_VEL
LIN {X 0,Y 573.066,Z 223.811,A -85,B 0,C 180,E1 -2004.338,E2 -2004.338} C_VEL
LIN {X 0,Y 573.03,Z 227.014,A -85,B 0,C 180,E1 -2006.986,E2 -2006.986} C_VEL
LIN {X 0,Y 573.037,Z 229.755,A -85,B 0,C 180,E1 -2009.453,E2 -2009.453} C_VEL
LIN {X 0,Y 572.942,Z 232.74,A -85,B 0,C 180,E1 -2012.181,E2 -2012.181} C_VEL
LIN {X 0,Y 572.936,Z 235.958,A -85,B 0,C 180,E1 -2014.73,E2 -2014.73} C_VEL
LIN {X 0,Y 572.89,Z 240.022,A -85,B 0,C 180,E1 -2017.832,E2 -2017.832} C_VEL
LIN {X 0,Y 572.923,Z 243.687,A -85,B 0,C 180,E1 -2020.594,E2 -2020.594} C_VEL
LIN {X 0,Y 573.837,Z 250.462,A -85,B 0,C 180,E1 -2020.761,E2 -2020.761} C_VEL
LIN {X 0,Y 573.73,Z 262.578,A -85,B 0,C 180,E1 -2021.119,E2 -2021.119} C_VEL
LIN {X 0,Y 573.591,Z 275.101,A -85,B 0,C 180,E1 -2021.635,E2 -2021.635} C_VEL
LIN {X 0,Y 573.481,Z 286.79,A -85,B 0,C 180,E1 -2022.276,E2 -2022.276} C_VEL
LIN {X 0,Y 573.383,Z 298.124,A -85,B 0,C 180,E1 -2023.065,E2 -2023.065} C_VEL
LIN {X 0,Y 573.288,Z 307.331,A -85,B 0,C 180,E1 -2023.855,E2 -2023.855} C_VEL
LIN {X 0,Y 573.165,Z 316.725,A -85,B 0,C 180,E1 -2024.849,E2 -2024.849} C_VEL
LIN {X 0,Y 573.108,Z 324.359,A -85,B 0,C 180,E1 -2025.842,E2 -2025.842} C_VEL
LIN {X 0,Y 573.042,Z 331.69,A -85,B 0,C 180,E1 -2027.028,E2 -2027.028} C_VEL
LIN {X 0,Y 573.026,Z 336.575,A -85,B 0,C 180,E1 -2028.032,E2 -2028.032} C_VEL
LIN {X 0,Y 573.004,Z 340.263,A -85,B 0,C 180,E1 -2028.991,E2 -2028.991} C_VEL
LIN {X 0,Y 572.95,Z 344.1,A -85,B 0,C 180,E1 -2030.369,E2 -2030.369} C_VEL
LIN {X 0,Y 572.939,Z 346.28,A -85,B 0,C 180,E1 -2031.724,E2 -2031.724} C_VEL
LIN {X 0,Y 572.952,Z 347,A -85,B 0,C 180,E1 -2033.056,E2 -2033.056} C_VEL
LIN {X 0,Y 572.92,Z 346.577,A -85,B 0,C 180,E1 -2034.056,E2 -2034.056} C_VEL
LIN {X 0,Y 572.954,Z 345.016,A -85,B 0,C 180,E1 -2035.266,E2 -2035.266} C_VEL
LIN {X 0,Y 572.973,Z 342.091,A -85,B 0,C 180,E1 -2036.517,E2 -2036.517} C_VEL
LIN {X 0,Y 572.988,Z 337.595,A -85,B 0,C 180,E1 -2037.811,E2 -2037.811} C_VEL
LIN {X 0,Y 573.052,Z 332.03,A -85,B 0,C 180,E1 -2038.997,E2 -2038.997} C_VEL
LIN {X 0,Y 573.107,Z 324.675,A -85,B 0,C 180,E1 -2040.203,E2 -2040.203} C_VEL
LIN {X 0,Y 573.159,Z 316.803,A -85,B 0,C 180,E1 -2041.232,E2 -2041.232} C_VEL
LIN {X 0,Y 573.3,Z 307.307,A -85,B 0,C 180,E1 -2042.237,E2 -2042.237} C_VEL
LIN {X 0,Y 573.398,Z 298.03,A -85,B 0,C 180,E1 -2043.032,E2 -2043.032} C_VEL
LIN {X 0,Y 573.494,Z 286.651,A -85,B 0,C 180,E1 -2043.822,E2 -2043.822} C_VEL
LIN {X 0,Y 573.623,Z 274.941,A -85,B 0,C 180,E1 -2044.462,E2 -2044.462} C_VEL
LIN {X 0,Y 573.717,Z 262.613,A -85,B 0,C 180,E1 -2044.97,E2 -2044.97} C_VEL
LIN {X 0,Y 573.834,Z 249.358,A -85,B 0,C 180,E1 -2045.356,E2 -2045.356} C_VEL
LIN {X 0,Y 572.958,Z 243.684,A -85,B 0,C 180,E1 -2045.497,E2 -2045.497} C_VEL
LIN {X 0,Y 572.943,Z 240.822,A -85,B 0,C 180,E1 -2047.651,E2 -2047.651} C_VEL
LIN {X 0,Y 572.978,Z 236.867,A -85,B 0,C 180,E1 -2050.661,E2 -2050.661} C_VEL
LIN {X 0,Y 572.975,Z 233.057,A -85,B 0,C 180,E1 -2053.614,E2 -2053.614} C_VEL
LIN {X 0,Y 573.05,Z 230.545,A -85,B 0,C 180,E1 -2055.802,E2 -2055.802} C_VEL
LIN {X 0,Y 573.077,Z 227.026,A -85,B 0,C 180,E1 -2058.83,E2 -2058.83} C_VEL
LIN {X 0,Y 573.085,Z 223.772,A -85,B 0,C 180,E1 -2061.538,E2 -2061.538} C_VEL
LIN {X 0,Y 573.107,Z 221.278,A -85,B 0,C 180,E1 -2063.664,E2 -2063.664} C_VEL
LIN {X 0,Y 573.131,Z 218.811,A -85,B 0,C 180,E1 -2065.781,E2 -2065.781} C_VEL
LIN {X 0,Y 573.063,Z 217.176,A -85,B 0,C 180,E1 -2067.189,E2 -2067.189} C_VEL
LIN {X 0,Y 573.33,Z 217.072,A -85,B 0,C 180,E1 -2069.298,E2 -2069.298} C_VEL
LIN {X 0,Y 573.299,Z 217.073,A -85,B 0,C 180,E1 -2072.108,E2 -2072.108} C_VEL
LIN {X 0,Y 573.284,Z 217.076,A -85,B 0,C 180,E1 -2075.629,E2 -2075.629} C_VEL
LIN {X 0,Y 573.296,Z 217.075,A -85,B 0,C 180,E1 -2078.46,E2 -2078.46} C_VEL
LIN {X 0,Y 573.286,Z 217.076,A -85,B 0,C 180,E1 -2081.312,E2 -2081.312} C_VEL
LIN {X 0,Y 573.268,Z 217.08,A -85,B 0,C 180,E1 -2084.426,E2 -2084.426} C_VEL
LIN {X 0,Y 573.248,Z 217.08,A -85,B 0,C 180,E1 -2087.113,E2 -2087.113} C_VEL
LIN {X 0,Y 573.247,Z 217.083,A -85,B 0,C 180,E1 -2090.077,E2 -2090.077} C_VEL
LIN {X 0,Y 573.261,Z 217.079,A -85,B 0,C 180,E1 -2093.155,E2 -2093.155} C_VEL
LIN {X 0,Y 573.282,Z 217.076,A -85,B 0,C 180,E1 -2096.19,E2 -2096.19} C_VEL
LIN {X 0,Y 573.233,Z 217.082,A -85,B 0,C 180,E1 -2098.565,E2 -2098.565} C_VEL
LIN {X 0,Y 573.227,Z 217.083,A -85,B 0,C 180,E1 -2100.994,E2 -2100.994} C_VEL
LIN {X 0,Y 573.279,Z 217.077,A -85,B 0,C 180,E1 -2103.53,E2 -2103.53} C_VEL
LIN {X 0,Y 573.253,Z 217.082,A -85,B 0,C 180,E1 -2106.049,E2 -2106.049} C_VEL
LIN {X 0,Y 573.24,Z 217.082,A -85,B 0,C 180,E1 -2108.703,E2 -2108.703} C_VEL
LIN {X 0,Y 573.247,Z 217.081,A -85,B 0,C 180,E1 -2111.597,E2 -2111.597} C_VEL
LIN {X 0,Y 573.233,Z 217.083,A -85,B 0,C 180,E1 -2114.335,E2 -2114.335} C_VEL
LIN {X 0,Y 573.235,Z 217.083,A -85,B 0,C 180,E1 -2117.36,E2 -2117.36} C_VEL
LIN {X 0,Y 573.245,Z 217.08,A -85,B 0,C 180,E1 -2120.395,E2 -2120.395} C_VEL
LIN {X 0,Y 573.253,Z 217.081,A -85,B 0,C 180,E1 -2123.08,E2 -2123.08} C_VEL
LIN {X 0,Y 573.266,Z 217.08,A -85,B 0,C 180,E1 -2125.673,E2 -2125.673} C_VEL
LIN {X 0,Y 573.239,Z 217.082,A -85,B 0,C 180,E1 -2128.186,E2 -2128.186} C_VEL
LIN {X 0,Y 573.265,Z 217.078,A -85,B 0,C 180,E1 -2130.636,E2 -2130.636} C_VEL
LIN {X 0,Y 573.25,Z 217.079,A -85,B 0,C 180,E1 -2133.026,E2 -2133.026} C_VEL
LIN {X 0,Y 573.275,Z 217.076,A -85,B 0,C 180,E1 -2135.368,E2 -2135.368} C_VEL
LIN {X 0,Y 573.23,Z 217.083,A -85,B 0,C 180,E1 -2138.421,E2 -2138.421} C_VEL
LIN {X 0,Y 573.281,Z 217.076,A -85,B 0,C 180,E1 -2140.73,E2 -2140.73} C_VEL
LIN {X 0,Y 573.245,Z 217.081,A -85,B 0,C 180,E1 -2143.623,E2 -2143.623} C_VEL
LIN {X 0,Y 573.276,Z 217.077,A -85,B 0,C 180,E1 -2145.808,E2 -2145.808} C_VEL
LIN {X 0,Y 573.268,Z 217.078,A -85,B 0,C 180,E1 -2148.746,E2 -2148.746} C_VEL
LIN {X 0,Y 573.26,Z 217.079,A -85,B 0,C 180,E1 -2151.541,E2 -2151.541} C_VEL
LIN {X 0,Y 573.253,Z 217.08,A -85,B 0,C 180,E1 -2153.666,E2 -2153.666} C_VEL
LIN {X 0,Y 573.229,Z 217.083,A -85,B 0,C 180,E1 -2155.783,E2 -2155.783} C_VEL
LIN {X 0,Y 573.303,Z 217.074,A -85,B 0,C 180,E1 -2157.894,E2 -2157.894} C_VEL
LIN {X 0,Y 573.33,Z 217.07,A -85,B 0,C 180,E1 -2160.703,E2 -2160.703} C_VEL
LIN {X 0,Y 573.304,Z 217.072,A -85,B 0,C 180,E1 -2162.812,E2 -2162.812} C_VEL
LIN {X 0,Y 573.29,Z 217.078,A -85,B 0,C 180,E1 -2165.629,E2 -2165.629} C_VEL
LIN {X 0,Y 573.279,Z 217.078,A -85,B 0,C 180,E1 -2167.751,E2 -2167.751} C_VEL
LIN {X 0,Y 573.268,Z 217.077,A -85,B 0,C 180,E1 -2170.598,E2 -2170.598} C_VEL
LIN {X 0,Y 573.247,Z 217.081,A -85,B 0,C 180,E1 -2172.75,E2 -2172.75} C_VEL
LIN {X 0,Y 573.241,Z 217.083,A -85,B 0,C 180,E1 -2174.92,E2 -2174.92} C_VEL
LIN {X 0,Y 573.235,Z 217.082,A -85,B 0,C 180,E1 -2177.85,E2 -2177.85} C_VEL
LIN {X 0,Y 573.249,Z 217.08,A -85,B 0,C 180,E1 -2180.078,E2 -2180.078} C_VEL
LIN {X 0,Y 573.24,Z 217.081,A -85,B 0,C 180,E1 -2182.338,E2 -2182.338} C_VEL
LIN {X 0,Y 573.244,Z 217.081,A -85,B 0,C 180,E1 -2185.411,E2 -2185.411} C_VEL
LIN {X 0,Y 573.256,Z 217.079,A -85,B 0,C 180,E1 -2188.028,E2 -2188.028} C_VEL
LIN {X 0,Y 573.244,Z 217.08,A -85,B 0,C 180,E1 -2190.177,E2 -2190.177} C_VEL
LIN {X 0,Y 573.259,Z 217.079,A -85,B 0,C 180,E1 -2192.645,E2 -2192.645} C_VEL
LIN {X 0,Y 573.214,Z 217.086,A -85,B 0,C 180,E1 -2195.188,E2 -2195.188} C_VEL
LIN {X 0,Y 573.24,Z 217.082,A -85,B 0,C 180,E1 -2197.808,E2 -2197.808} C_VEL
LIN {X 0,Y 573.254,Z 217.079,A -85,B 0,C 180,E1 -2200.525,E2 -2200.525} C_VEL
LIN {X 0,Y 573.245,Z 217.083,A -85,B 0,C 180,E1 -2203.359,E2 -2203.359} C_VEL
LIN {X 0,Y 573.244,Z 217.082,A -85,B 0,C 180,E1 -2206.641,E2 -2206.641} C_VEL
LIN {X 0,Y 573.253,Z 217.08,A -85,B 0,C 180,E1 -2209.475,E2 -2209.475} C_VEL
LIN {X 0,Y 573.236,Z 217.083,A -85,B 0,C 180,E1 -2212.192,E2 -2212.192} C_VEL
LIN {X 0,Y 573.266,Z 217.161,A -85,B 0,C 180,E1 -2213.242,E2 -2213.242} C_VEL
LIN {X 0,Y 573.752,Z 221.795,A -85,B 0,C 180,E1 -2214.85,E2 -2214.85} C_VEL
LIN {X 0,Y 573.678,Z 229.53,A -85,B 0,C 180,E1 -2217.381,E2 -2217.381} C_VEL
LIN {X 0,Y 573.5,Z 237.317,A -85,B 0,C 180,E1 -2219.838,E2 -2219.838} C_VEL
LIN {X 0,Y 573.417,Z 246.769,A -85,B 0,C 180,E1 -2222.637,E2 -2222.637} C_VEL
LIN {X 0,Y 573.369,Z 256.199,A -85,B 0,C 180,E1 -2225.37,E2 -2225.37} C_VEL
LIN {X 0,Y 573.324,Z 266.927,A -85,B 0,C 180,E1 -2228.422,E2 -2228.422} C_VEL
LIN {X 0,Y 573.218,Z 277.518,A -85,B 0,C 180,E1 -2231.41,E2 -2231.41} C_VEL
LIN {X 0,Y 573.162,Z 288.109,A -85,B 0,C 180,E1 -2234.349,E2 -2234.349} C_VEL
LIN {X 0,Y 573.096,Z 297.376,A -85,B 0,C 180,E1 -2236.886,E2 -2236.886} C_VEL
LIN {X 0,Y 573.087,Z 299.528,A -85,B 0,C 180,E1 -2237.472,E2 -2237.472} C_VEL
LIN {X 0,Y 573.869,Z 306.334,A -85,B 0,C 180,E1 -2237.624,E2 -2237.624} C_VEL
LIN {X 0,Y 573.782,Z 318.475,A -85,B 0,C 180,E1 -2237.936,E2 -2237.936} C_VEL
LIN {X 0,Y 573.652,Z 330.301,A -85,B 0,C 180,E1 -2238.373,E2 -2238.373} C_VEL
LIN {X 0,Y 573.512,Z 342.471,A -85,B 0,C 180,E1 -2238.976,E2 -2238.976} C_VEL
LIN {X 0,Y 573.45,Z 353.472,A -85,B 0,C 180,E1 -2239.674,E2 -2239.674} C_VEL
LIN {X 0,Y 573.308,Z 363.639,A -85,B 0,C 180,E1 -2240.473,E2 -2240.473} C_VEL
LIN {X 0,Y 573.207,Z 372.78,A -85,B 0,C 180,E1 -2241.361,E2 -2241.361} C_VEL
LIN {X 0,Y 573.143,Z 381.684,A -85,B 0,C 180,E1 -2242.425,E2 -2242.425} C_VEL
LIN {X 0,Y 573.052,Z 388.405,A -85,B 0,C 180,E1 -2243.415,E2 -2243.415} C_VEL
LIN {X 0,Y 573.071,Z 393.676,A -85,B 0,C 180,E1 -2244.369,E2 -2244.369} C_VEL
LIN {X 0,Y 573.029,Z 398.369,A -85,B 0,C 180,E1 -2245.427,E2 -2245.427} C_VEL
LIN {X 0,Y 573.022,Z 401.955,A -85,B 0,C 180,E1 -2246.483,E2 -2246.483} C_VEL
LIN {X 0,Y 572.959,Z 403.806,A -85,B 0,C 180,E1 -2247.187,E2 -2247.187} C_VEL
LIN {X 0,Y 572.94,Z 405.197,A -85,B 0,C 180,E1 -2247.89,E2 -2247.89} C_VEL
LIN {X 0,Y 572.941,Z 406.784,A -85,B 0,C 180,E1 -2249.296,E2 -2249.296} C_VEL
LIN {X 0,Y 572.938,Z 407,A -85,B 0,C 180,E1 -2249.999,E2 -2249.999} C_VEL
LIN {X 0,Y 572.946,Z 406.187,A -85,B 0,C 180,E1 -2251.405,E2 -2251.405} C_VEL
LIN {X 0,Y 572.94,Z 405.201,A -85,B 0,C 180,E1 -2252.108,E2 -2252.108} C_VEL
LIN {X 0,Y 572.959,Z 403.812,A -85,B 0,C 180,E1 -2252.812,E2 -2252.812} C_VEL
LIN {X 0,Y 573.015,Z 400.898,A -85,B 0,C 180,E1 -2253.867,E2 -2253.867} C_VEL
LIN {X 0,Y 572.963,Z 396.952,A -85,B 0,C 180,E1 -2254.925,E2 -2254.925} C_VEL
LIN {X 0,Y 573.065,Z 390.881,A -85,B 0,C 180,E1 -2256.159,E2 -2256.159} C_VEL
LIN {X 0,Y 573.119,Z 384.243,A -85,B 0,C 180,E1 -2257.22,E2 -2257.22} C_VEL
LIN {X 0,Y 573.201,Z 375.997,A -85,B 0,C 180,E1 -2258.282,E2 -2258.282} C_VEL
LIN {X 0,Y 573.287,Z 367.546,A -85,B 0,C 180,E1 -2259.17,E2 -2259.17} C_VEL
LIN {X 0,Y 573.43,Z 357.108,A -85,B 0,C 180,E1 -2260.057,E2 -2260.057} C_VEL
LIN {X 0,Y 573.512,Z 345.543,A -85,B 0,C 180,E1 -2260.847,E2 -2260.847} C_VEL
LIN {X 0,Y 573.609,Z 333.9,A -85,B 0,C 180,E1 -2261.465,E2 -2261.465} C_VEL
LIN {X 0,Y 573.755,Z 321.193,A -85,B 0,C 180,E1 -2261.973,E2 -2261.973} C_VEL
LIN {X 0,Y 573.868,Z 308.549,A -85,B 0,C 180,E1 -2262.33,E2 -2262.33} C_VEL
LIN {X 0,Y 573.575,Z 302.689,A -85,B 0,C 180,E1 -2262.454,E2 -2262.454} C_VEL
LIN {X 0,Y 573.085,Z 299.533,A -85,B 0,C 180,E1 -2262.527,E2 -2262.527} C_VEL
LIN {X 0,Y 573.158,Z 289.438,A -85,B 0,C 180,E1 -2265.285,E2 -2265.285} C_VEL
LIN {X 0,Y 573.217,Z 278.847,A -85,B 0,C 180,E1 -2268.218,E2 -2268.218} C_VEL
LIN {X 0,Y 573.297,Z 269.58,A -85,B 0,C 180,E1 -2270.824,E2 -2270.824} C_VEL
LIN {X 0,Y 573.313,Z 261.216,A -85,B 0,C 180,E1 -2273.162,E2 -2273.162} C_VEL
LIN {X 0,Y 573.357,Z 251.692,A -85,B 0,C 180,E1 -2275.794,E2 -2275.794} C_VEL
LIN {X 0,Y 573.421,Z 242.43,A -85,B 0,C 180,E1 -2278.554,E2 -2278.554} C_VEL
LIN {X 0,Y 573.62,Z 233.31,A -85,B 0,C 180,E1 -2281.379,E2 -2281.379} C_VEL
LIN {X 0,Y 573.701,Z 224.285,A -85,B 0,C 180,E1 -2284.298,E2 -2284.298} C_VEL
LIN {X 0,Y 573.598,Z 219.208,A -85,B 0,C 180,E1 -2286.034,E2 -2286.034} C_VEL
LIN {X 0,Y 573.262,Z 217.081,A -85,B 0,C 180,E1 -2286.811,E2 -2286.811} C_VEL
LIN {X 0,Y 573.248,Z 217.083,A -85,B 0,C 180,E1 -2289.606,E2 -2289.606} C_VEL
LIN {X 0,Y 573.242,Z 217.081,A -85,B 0,C 180,E1 -2292.641,E2 -2292.641} C_VEL
LIN {X 0,Y 573.213,Z 217.087,A -85,B 0,C 180,E1 -2295.325,E2 -2295.325} C_VEL
LIN {X 0,Y 573.239,Z 217.084,A -85,B 0,C 180,E1 -2297.599,E2 -2297.599} C_VEL
LIN {X 0,Y 573.241,Z 217.081,A -85,B 0,C 180,E1 -2300.392,E2 -2300.392} C_VEL
LIN {X 0,Y 573.251,Z 217.081,A -85,B 0,C 180,E1 -2303.077,E2 -2303.077} C_VEL
LIN {X 0,Y 573.272,Z 217.08,A -85,B 0,C 180,E1 -2305.671,E2 -2305.671} C_VEL
LIN {X 0,Y 573.238,Z 217.082,A -85,B 0,C 180,E1 -2308.184,E2 -2308.184} C_VEL
LIN {X 0,Y 573.264,Z 217.078,A -85,B 0,C 180,E1 -2310.633,E2 -2310.633} C_VEL
LIN {X 0,Y 573.25,Z 217.08,A -85,B 0,C 180,E1 -2313.023,E2 -2313.023} C_VEL
LIN {X 0,Y 573.272,Z 217.077,A -85,B 0,C 180,E1 -2315.365,E2 -2315.365} C_VEL
LIN {X 0,Y 573.226,Z 217.083,A -85,B 0,C 180,E1 -2318.418,E2 -2318.418} C_VEL
LIN {X 0,Y 573.275,Z 217.077,A -85,B 0,C 180,E1 -2320.727,E2 -2320.727} C_VEL
LIN {X 0,Y 573.25,Z 217.082,A -85,B 0,C 180,E1 -2323.621,E2 -2323.621} C_VEL
LIN {X 0,Y 573.271,Z 217.078,A -85,B 0,C 180,E1 -2325.806,E2 -2325.806} C_VEL
LIN {X 0,Y 573.258,Z 217.079,A -85,B 0,C 180,E1 -2328.744,E2 -2328.744} C_VEL
